LIN {X 0,Y 446.131,Z 914.259,A -85,B 0,C 180,E1 18585.632,E2 18585.632} C_VEL
LIN {X 0,Y 452.831,Z 893.973,A -85,B 0,C 180,E1 18583.695,E2 18583.695} C_VEL
LIN {X 0,Y 459.309,Z 872.522,A -85,B 0,C 180,E1 18581.967,E2 18581.967} C_VEL
LIN {X 0,Y 464.542,Z 853.932,A -85,B 0,C 180,E1 18580.675,E2 18580.675} C_VEL
LIN {X 0,Y 469.911,Z 833.178,A -85,B 0,C 180,E1 18579.43,E2 18579.43} C_VEL
LIN {X 0,Y 475.402,Z 809.084,A -85,B 0,C 180,E1 18578.228,E2 18578.228} C_VEL
LIN {X 0,Y 479.6,Z 787.75,A -85,B 0,C 180,E1 18577.351,E2 18577.351} C_VEL
LIN {X 0,Y 483.367,Z 765.529,A -85,B 0,C 180,E1 18576.603,E2 18576.603} C_VEL
LIN {X 0,Y 487.105,Z 737.581,A -85,B 0,C 180,E1 18575.887,E2 18575.887} C_VEL
LIN {X 0,Y 489.19,Z 714.963,A -85,B 0,C 180,E1 18575.454,E2 18575.454} C_VEL
LIN {X 0,Y 502.118,Z 484.551,A -85,B 0,C 180,E1 18571.853,E2 18571.853} C_VEL
LIN {X 0,Y 505.42,Z 425.189,A -85,B 0,C 180,E1 18570.906,E2 18570.906} C_VEL
LIN {X 0,Y 497.545,Z 411.726,A -85,B 0,C 180,E1 18569.067,E2 18569.067} C_VEL
LIN {X 0,Y 488.892,Z 397.653,A -85,B 0,C 180,E1 18566.872,E2 18566.872} C_VEL
LIN {X 0,Y 478.631,Z 382.114,A -85,B 0,C 180,E1 18563.974,E2 18563.974} C_VEL
LIN {X 0,Y 470.083,Z 371.062,A -85,B 0,C 180,E1 18561.264,E2 18561.264} C_VEL
LIN {X 0,Y 465.83,Z 365.703,A -85,B 0,C 180,E1 18559.759,E2 18559.759} C_VEL
LIN {X 0,Y 461.713,Z 360.509,A -85,B 0,C 180,E1 18558.171,E2 18558.171} C_VEL
LIN {X 0,Y 457.361,Z 355.125,A -85,B 0,C 180,E1 18556.316,E2 18556.316} C_VEL
LIN {X 0,Y 453.894,Z 351.057,A -85,B 0,C 180,E1 18554.675,E2 18554.675} C_VEL
LIN {X 0,Y 452.721,Z 349.402,A -85,B 0,C 180,E1 18554.061,E2 18554.061} C_VEL
LIN {X 0,Y 449.237,Z 345.797,A -85,B 0,C 180,E1 18552.142,E2 18552.142} C_VEL
LIN {X 0,Y 447.81,Z 343.423,A -85,B 0,C 180,E1 18551.201,E2 18551.201} C_VEL
LIN {X 0,Y 444.369,Z 340.419,A -85,B 0,C 180,E1 18548.801,E2 18548.801} C_VEL
LIN {X 0,Y 442.614,Z 337.176,A -85,B 0,C 180,E1 18547.137,E2 18547.137} C_VEL
LIN {X 0,Y 438.09,Z 332.937,A -85,B 0,C 180,E1 18539.346,E2 18539.346} C_VEL
LIN {X 0,Y 438.15,Z 333.065,A -85,B 0,C 180,E1 18536.991,E2 18536.991} C_VEL
LIN {X 0,Y 442.91,Z 337.557,A -85,B 0,C 180,E1 18529.398,E2 18529.398} C_VEL
LIN {X 0,Y 444.805,Z 340.967,A -85,B 0,C 180,E1 18527.669,E2 18527.669} C_VEL
LIN {X 0,Y 448.152,Z 343.843,A -85,B 0,C 180,E1 18525.397,E2 18525.397} C_VEL
LIN {X 0,Y 450.898,Z 347.851,A -85,B 0,C 180,E1 18523.709,E2 18523.709} C_VEL
LIN {X 0,Y 453.392,Z 350.187,A -85,B 0,C 180,E1 18522.414,E2 18522.414} C_VEL
LIN {X 0,Y 456.634,Z 354.467,A -85,B 0,C 180,E1 18520.825,E2 18520.825} C_VEL
LIN {X 0,Y 458.34,Z 356.318,A -85,B 0,C 180,E1 18520.07,E2 18520.07} C_VEL
LIN {X 0,Y 462.075,Z 360.858,A -85,B 0,C 180,E1 18518.509,E2 18518.509} C_VEL
LIN {X 0,Y 467.83,Z 368.146,A -85,B 0,C 180,E1 18516.342,E2 18516.342} C_VEL
LIN {X 0,Y 472.295,Z 373.974,A -85,B 0,C 180,E1 18514.815,E2 18514.815} C_VEL
LIN {X 0,Y 479.579,Z 383.444,A -85,B 0,C 180,E1 18512.563,E2 18512.563} C_VEL
LIN {X 0,Y 489.38,Z 397.087,A -85,B 0,C 180,E1 18509.86,E2 18509.86} C_VEL
LIN {X 0,Y 497.663,Z 409.437,A -85,B 0,C 180,E1 18507.796,E2 18507.796} C_VEL
LIN {X 0,Y 505.573,Z 422.879,A -85,B 0,C 180,E1 18505.951,E2 18505.951} C_VEL
LIN {X 0,Y 493.861,Z 629.815,A -85,B 0,C 180,E1 18502.723,E2 18502.723} C_VEL
LIN {X 0,Y 489.029,Z 714.247,A -85,B 0,C 180,E1 18501.386,E2 18501.386} C_VEL
LIN {X 0,Y 486.062,Z 742.57,A -85,B 0,C 180,E1 18500.783,E2 18500.783} C_VEL
LIN {X 0,Y 483.078,Z 763.5,A -85,B 0,C 180,E1 18500.191,E2 18500.191} C_VEL
LIN {X 0,Y 479.517,Z 784.275,A -85,B 0,C 180,E1 18499.469,E2 18499.469} C_VEL
LIN {X 0,Y 474.318,Z 810.058,A -85,B 0,C 180,E1 18498.357,E2 18498.357} C_VEL
LIN {X 0,Y 469.237,Z 831.534,A -85,B 0,C 180,E1 18497.223,E2 18497.223} C_VEL
LIN {X 0,Y 464.133,Z 851.066,A -85,B 0,C 180,E1 18496.016,E2 18496.016} C_VEL
LIN {X 0,Y 457.617,Z 873.85,A -85,B 0,C 180,E1 18494.362,E2 18494.362} C_VEL
LIN {X 0,Y 451.329,Z 893.778,A -85,B 0,C 180,E1 18492.648,E2 18492.648} C_VEL
LIN {X 0,Y 445.384,Z 911.684,A -85,B 0,C 180,E1 18490.875,E2 18490.875} C_VEL
LIN {X 0,Y 438.182,Z 932.354,A -85,B 0,C 180,E1 18488.492,E2 18488.492} C_VEL
LIN {X 0,Y 432.293,Z 948.557,A -85,B 0,C 180,E1 18486.308,E2 18486.308} C_VEL
LIN {X 0,Y 426.626,Z 963.981,A -85,B 0,C 180,E1 18483.934,E2 18483.934} C_VEL
LIN {X 0,Y 420.149,Z 981.509,A -85,B 0,C 180,E1 18480.781,E2 18480.781} C_VEL
LIN {X 0,Y 415.589,Z 994.103,A -85,B 0,C 180,E1 18478.136,E2 18478.136} C_VEL
LIN {X 0,Y 411.172,Z 1006.966,A -85,B 0,C 180,E1 18475.032,E2 18475.032} C_VEL
LIN {X 0,Y 407.325,Z 1018.86,A -85,B 0,C 180,E1 18471.605,E2 18471.605} C_VEL
LIN {X 0,Y 404.734,Z 1027.798,A -85,B 0,C 180,E1 18468.584,E2 18468.584} C_VEL
LIN {X 0,Y 402.535,Z 1036.804,A -85,B 0,C 180,E1 18464.971,E2 18464.971} C_VEL
LIN {X 0,Y 401.176,Z 1043.635,A -85,B 0,C 180,E1 18461.501,E2 18461.501} C_VEL
LIN {X 0,Y 400.461,Z 1048.425,A -85,B 0,C 180,E1 18458.471,E2 18458.471} C_VEL
LIN {X 0,Y 400.088,Z 1052.26,A -85,B 0,C 180,E1 18455.306,E2 18455.306} C_VEL
LIN {X 0,Y 399.924,Z 1055.14,A -85,B 0,C 180,E1 18451.719,E2 18451.719} C_VEL
LIN {X 0,Y 399.904,Z 1056.343,A -85,B 0,C 180,E1 18448.567,E2 18448.567} C_VEL
LIN {X 0,Y 399.903,Z 1056.481,A -85,B 0,C 180,E1 18447.693,E2 18447.693} C_VEL
LIN {X 0,Y 398.901,Z 1056.59,A -85,B 0,C 180,E1 18446.59,E2 18446.59} C_VEL
LIN {X 0,Y 392.465,Z 1056.003,A -85,B 0,C 180,E1 18443.478,E2 18443.478} C_VEL
LIN {X 0,Y 391.928,Z 1055.619,A -85,B 0,C 180,E1 18442.666,E2 18442.666} C_VEL
LIN {X 0,Y 392.038,Z 1053.632,A -85,B 0,C 180,E1 18439.567,E2 18439.567} C_VEL
LIN {X 0,Y 392.422,Z 1049.847,A -85,B 0,C 180,E1 18435.841,E2 18435.841} C_VEL
LIN {X 0,Y 393.228,Z 1044.792,A -85,B 0,C 180,E1 18432.387,E2 18432.387} C_VEL
LIN {X 0,Y 394.417,Z 1039.146,A -85,B 0,C 180,E1 18429.303,E2 18429.303} C_VEL
LIN {X 0,Y 396.415,Z 1031.684,A -85,B 0,C 180,E1 18425.936,E2 18425.936} C_VEL
LIN {X 0,Y 399.69,Z 1021.249,A -85,B 0,C 180,E1 18422.108,E2 18422.108} C_VEL
LIN {X 0,Y 403.089,Z 1011.528,A -85,B 0,C 180,E1 18419.104,E2 18419.104} C_VEL
LIN {X 0,Y 407.809,Z 999.269,A -85,B 0,C 180,E1 18415.842,E2 18415.842} C_VEL
LIN {X 0,Y 413.485,Z 984.893,A -85,B 0,C 180,E1 18412.63,E2 18412.63} C_VEL
LIN {X 0,Y 418.923,Z 971.568,A -85,B 0,C 180,E1 18410.055,E2 18410.055} C_VEL
LIN {X 0,Y 425.983,Z 954.445,A -85,B 0,C 180,E1 18407.196,E2 18407.196} C_VEL
LIN {X 0,Y 432.891,Z 937.105,A -85,B 0,C 180,E1 18404.744,E2 18404.744} C_VEL
LIN {X 0,Y 439.213,Z 920.922,A -85,B 0,C 180,E1 18402.752,E2 18402.752} C_VEL
LIN {X 0,Y 446.85,Z 900.493,A -85,B 0,C 180,E1 18400.582,E2 18400.582} C_VEL
LIN {X 0,Y 453.657,Z 880.878,A -85,B 0,C 180,E1 18398.819,E2 18398.819} C_VEL
LIN {X 0,Y 459.787,Z 862.035,A -85,B 0,C 180,E1 18397.354,E2 18397.354} C_VEL
LIN {X 0,Y 466.454,Z 839.808,A -85,B 0,C 180,E1 18395.877,E2 18395.877} C_VEL
LIN {X 0,Y 472.255,Z 817.735,A -85,B 0,C 180,E1 18394.659,E2 18394.659} C_VEL
LIN {X 0,Y 476.724,Z 798.729,A -85,B 0,C 180,E1 18393.767,E2 18393.767} C_VEL
LIN {X 0,Y 481.183,Z 777.074,A -85,B 0,C 180,E1 18392.913,E2 18392.913} C_VEL
LIN {X 0,Y 485.71,Z 750.138,A -85,B 0,C 180,E1 18392.076,E2 18392.076} C_VEL
LIN {X 0,Y 488.616,Z 727.847,A -85,B 0,C 180,E1 18391.55,E2 18391.55} C_VEL
LIN {X 0,Y 490.902,Z 702.791,A -85,B 0,C 180,E1 18391.093,E2 18391.093} C_VEL
LIN {X 0,Y 505.255,Z 471.196,A -85,B 0,C 180,E1 18387.473,E2 18387.473} C_VEL
LIN {X 0,Y 507.793,Z 430.464,A -85,B 0,C 180,E1 18386.82,E2 18386.82} C_VEL
LIN {X 0,Y 500.137,Z 417.918,A -85,B 0,C 180,E1 18384.762,E2 18384.762} C_VEL
LIN {X 0,Y 492.623,Z 406.949,A -85,B 0,C 180,E1 18382.558,E2 18382.558} C_VEL
LIN {X 0,Y 485.385,Z 396.927,A -85,B 0,C 180,E1 18380.185,E2 18380.185} C_VEL
LIN {X 0,Y 480.887,Z 391.016,A -85,B 0,C 180,E1 18378.55,E2 18378.55} C_VEL
LIN {X 0,Y 477.714,Z 386.768,A -85,B 0,C 180,E1 18377.291,E2 18377.291} C_VEL
LIN {X 0,Y 474.093,Z 382.002,A -85,B 0,C 180,E1 18375.725,E2 18375.725} C_VEL
LIN {X 0,Y 469.843,Z 376.609,A -85,B 0,C 180,E1 18373.664,E2 18373.664} C_VEL
LIN {X 0,Y 466.423,Z 372.307,A -85,B 0,C 180,E1 18371.751,E2 18371.751} C_VEL
LIN {X 0,Y 465.453,Z 371.035,A -85,B 0,C 180,E1 18371.148,E2 18371.148} C_VEL
LIN {X 0,Y 462.123,Z 367.252,A -85,B 0,C 180,E1 18368.837,E2 18368.837} C_VEL
LIN {X 0,Y 461.146,Z 365.386,A -85,B 0,C 180,E1 18367.977,E2 18367.977} C_VEL
LIN {X 0,Y 457.851,Z 362.35,A -85,B 0,C 180,E1 18364.635,E2 18364.635} C_VEL
LIN {X 0,Y 456.621,Z 359.617,A -85,B 0,C 180,E1 18362.385,E2 18362.385} C_VEL
LIN {X 0,Y 455.677,Z 358.962,A -85,B 0,C 180,E1 18358.365,E2 18358.365} C_VEL
LIN {X 0,Y 456.743,Z 359.705,A -85,B 0,C 180,E1 18354.472,E2 18354.472} C_VEL
LIN {X 0,Y 459.197,Z 364.086,A -85,B 0,C 180,E1 18350.854,E2 18350.854} C_VEL
LIN {X 0,Y 461.418,Z 365.771,A -85,B 0,C 180,E1 18348.88,E2 18348.88} C_VEL
LIN {X 0,Y 464.109,Z 369.819,A -85,B 0,C 180,E1 18346.799,E2 18346.799} C_VEL
LIN {X 0,Y 466.134,Z 371.817,A -85,B 0,C 180,E1 18345.528,E2 18345.528} C_VEL
LIN {X 0,Y 469.371,Z 376.177,A -85,B 0,C 180,E1 18343.668,E2 18343.668} C_VEL
LIN {X 0,Y 470.895,Z 377.833,A -85,B 0,C 180,E1 18342.897,E2 18342.897} C_VEL
LIN {X 0,Y 475.393,Z 383.739,A -85,B 0,C 180,E1 18340.788,E2 18340.788} C_VEL
LIN {X 0,Y 480.025,Z 389.872,A -85,B 0,C 180,E1 18338.878,E2 18338.878} C_VEL
LIN {X 0,Y 484.61,Z 396.005,A -85,B 0,C 180,E1 18337.176,E2 18337.176} C_VEL
LIN {X 0,Y 491.704,Z 406.708,A -85,B 0,C 180,E1 18334.784,E2 18334.784} C_VEL
LIN {X 0,Y 499.013,Z 418.174,A -85,B 0,C 180,E1 18332.59,E2 18332.59} C_VEL
LIN {X 0,Y 507.826,Z 432.949,A -85,B 0,C 180,E1 18330.199,E2 18330.199} C_VEL
LIN {X 0,Y 493.862,Z 655.807,A -85,B 0,C 180,E1 18326.718,E2 18326.718} C_VEL
LIN {X 0,Y 489.698,Z 720.789,A -85,B 0,C 180,E1 18325.679,E2 18325.679} C_VEL
LIN {X 0,Y 486.513,Z 748.326,A -85,B 0,C 180,E1 18325.1,E2 18325.1} C_VEL
LIN {X 0,Y 483.152,Z 769.669,A -85,B 0,C 180,E1 18324.517,E2 18324.517} C_VEL
LIN {X 0,Y 478.792,Z 792.887,A -85,B 0,C 180,E1 18323.717,E2 18323.717} C_VEL
LIN {X 0,Y 473.1,Z 818.082,A -85,B 0,C 180,E1 18322.624,E2 18322.624} C_VEL
LIN {X 0,Y 467.737,Z 838.822,A -85,B 0,C 180,E1 18321.532,E2 18321.532} C_VEL
LIN {X 0,Y 461.508,Z 860.63,A -85,B 0,C 180,E1 18320.179,E2 18320.179} C_VEL
LIN {X 0,Y 454.148,Z 883.618,A -85,B 0,C 180,E1 18318.466,E2 18318.466} C_VEL
LIN {X 0,Y 447.905,Z 901.761,A -85,B 0,C 180,E1 18316.885,E2 18316.885} C_VEL
LIN {X 0,Y 440.681,Z 921.68,A -85,B 0,C 180,E1 18314.882,E2 18314.882} C_VEL
LIN {X 0,Y 433.14,Z 941.135,A -85,B 0,C 180,E1 18312.561,E2 18312.561} C_VEL
LIN {X 0,Y 427.011,Z 956.58,A -85,B 0,C 180,E1 18310.438,E2 18310.438} C_VEL
LIN {X 0,Y 420.13,Z 973.846,A -85,B 0,C 180,E1 18307.709,E2 18307.709} C_VEL
LIN {X 0,Y 413.758,Z 989.517,A -85,B 0,C 180,E1 18304.772,E2 18304.772} C_VEL
LIN {X 0,Y 408.784,Z 1002.114,A -85,B 0,C 180,E1 18302.058,E2 18302.058} C_VEL
LIN {X 0,Y 403.583,Z 1016.015,A -85,B 0,C 180,E1 18298.565,E2 18298.565} C_VEL
LIN {X 0,Y 399.775,Z 1026.875,A -85,B 0,C 180,E1 18295.321,E2 18295.321} C_VEL
LIN {X 0,Y 396.982,Z 1035.848,A -85,B 0,C 180,E1 18292.198,E2 18292.198} C_VEL
LIN {X 0,Y 394.459,Z 1045.402,A -85,B 0,C 180,E1 18288.167,E2 18288.167} C_VEL
LIN {X 0,Y 393.21,Z 1051.386,A -85,B 0,C 180,E1 18285.033,E2 18285.033} C_VEL
LIN {X 0,Y 392.45,Z 1056.21,A -85,B 0,C 180,E1 18281.91,E2 18281.91} C_VEL
LIN {X 0,Y 392.045,Z 1060.472,A -85,B 0,C 180,E1 18278.279,E2 18278.279} C_VEL
LIN {X 0,Y 391.909,Z 1063.031,A -85,B 0,C 180,E1 18274.683,E2 18274.683} C_VEL
LIN {X 0,Y 391.902,Z 1064.068,A -85,B 0,C 180,E1 18271.755,E2 18271.755} C_VEL
LIN {X 0,Y 391.912,Z 1064.138,A -85,B 0,C 180,E1 18268.977,E2 18268.977} C_VEL
LIN {X 0,Y 391.912,Z 1063.308,A -85,B 0,C 180,E1 18266.197,E2 18266.197} C_VEL
LIN {X 0,Y 391.968,Z 1061.457,A -85,B 0,C 180,E1 18263.261,E2 18263.261} C_VEL
LIN {X 0,Y 392.158,Z 1058.434,A -85,B 0,C 180,E1 18260.164,E2 18260.164} C_VEL
LIN {X 0,Y 392.806,Z 1053.089,A -85,B 0,C 180,E1 18256.306,E2 18256.306} C_VEL
LIN {X 0,Y 393.863,Z 1047.064,A -85,B 0,C 180,E1 18253.026,E2 18253.026} C_VEL
LIN {X 0,Y 395.366,Z 1040.429,A -85,B 0,C 180,E1 18250.037,E2 18250.037} C_VEL
LIN {X 0,Y 397.97,Z 1030.979,A -85,B 0,C 180,E1 18246.454,E2 18246.454} C_VEL
LIN {X 0,Y 401.376,Z 1019.976,A -85,B 0,C 180,E1 18243.039,E2 18243.039} C_VEL
LIN {X 0,Y 404.921,Z 1009.552,A -85,B 0,C 180,E1 18240.242,E2 18240.242} C_VEL
LIN {X 0,Y 409.991,Z 995.753,A -85,B 0,C 180,E1 18237.03,E2 18237.03} C_VEL
LIN {X 0,Y 415.607,Z 980.582,A -85,B 0,C 180,E1 18234.054,E2 18234.054} C_VEL
LIN {X 0,Y 420.867,Z 966.706,A -85,B 0,C 180,E1 18231.678,E2 18231.678} C_VEL
LIN {X 0,Y 427.585,Z 949.121,A -85,B 0,C 180,E1 18229.054,E2 18229.054} C_VEL
LIN {X 0,Y 434.403,Z 930.424,A -85,B 0,C 180,E1 18226.692,E2 18226.692} C_VEL
LIN {X 0,Y 440.243,Z 913.957,A -85,B 0,C 180,E1 18224.878,E2 18224.878} C_VEL
LIN {X 0,Y 447.095,Z 893.834,A -85,B 0,C 180,E1 18222.946,E2 18222.946} C_VEL
LIN {X 0,Y 453.756,Z 872.421,A -85,B 0,C 180,E1 18221.214,E2 18221.214} C_VEL
LIN {X 0,Y 459.049,Z 854.175,A -85,B 0,C 180,E1 18219.94,E2 18219.94} C_VEL
LIN {X 0,Y 464.488,Z 833.744,A -85,B 0,C 180,E1 18218.708,E2 18218.708} C_VEL
LIN {X 0,Y 470.469,Z 808.208,A -85,B 0,C 180,E1 18217.433,E2 18217.433} C_VEL
LIN {X 0,Y 474.742,Z 786.949,A -85,B 0,C 180,E1 18216.564,E2 18216.564} C_VEL
LIN {X 0,Y 478.746,Z 763.73,A -85,B 0,C 180,E1 18215.789,E2 18215.789} C_VEL
LIN {X 0,Y 482.363,Z 736.862,A -85,B 0,C 180,E1 18215.114,E2 18215.114} C_VEL
LIN {X 0,Y 484.457,Z 714.471,A -85,B 0,C 180,E1 18214.686,E2 18214.686} C_VEL
LIN {X 0,Y 497.803,Z 483.887,A -85,B 0,C 180,E1 18211.07,E2 18211.07} C_VEL
LIN {X 0,Y 500.96,Z 429.227,A -85,B 0,C 180,E1 18210.197,E2 18210.197} C_VEL
LIN {X 0,Y 491.432,Z 413.006,A -85,B 0,C 180,E1 18207.87,E2 18207.87} C_VEL
LIN {X 0,Y 483.386,Z 400.09,A -85,B 0,C 180,E1 18205.714,E2 18205.714} C_VEL
LIN {X 0,Y 475.776,Z 388.58,A -85,B 0,C 180,E1 18203.469,E2 18203.469} C_VEL
LIN {X 0,Y 468.088,Z 378.415,A -85,B 0,C 180,E1 18200.965,E2 18200.965} C_VEL
LIN {X 0,Y 463.74,Z 372.888,A -85,B 0,C 180,E1 18199.393,E2 18199.393} C_VEL
LIN {X 0,Y 459.847,Z 367.901,A -85,B 0,C 180,E1 18197.854,E2 18197.854} C_VEL
LIN {X 0,Y 455.606,Z 362.601,A -85,B 0,C 180,E1 18196.004,E2 18196.004} C_VEL
LIN {X 0,Y 452.077,Z 358.219,A -85,B 0,C 180,E1 18194.277,E2 18194.277} C_VEL
LIN {X 0,Y 451.026,Z 356.927,A -85,B 0,C 180,E1 18193.722,E2 18193.722} C_VEL
LIN {X 0,Y 447.649,Z 353.179,A -85,B 0,C 180,E1 18191.793,E2 18191.793} C_VEL
LIN {X 0,Y 446.436,Z 351.192,A -85,B 0,C 180,E1 18190.975,E2 18190.975} C_VEL
LIN {X 0,Y 443.006,Z 347.999,A -85,B 0,C 180,E1 18188.502,E2 18188.502} C_VEL
LIN {X 0,Y 441.501,Z 345.069,A -85,B 0,C 180,E1 18187.025,E2 18187.025} C_VEL
LIN {X 0,Y 437.114,Z 340.88,A -85,B 0,C 180,E1 18179.345,E2 18179.345} C_VEL
LIN {X 0,Y 437.175,Z 341.01,A -85,B 0,C 180,E1 18176.985,E2 18176.985} C_VEL
LIN {X 0,Y 441.727,Z 345.427,A -85,B 0,C 180,E1 18169.567,E2 18169.567} C_VEL
LIN {X 0,Y 443.835,Z 349.051,A -85,B 0,C 180,E1 18167.642,E2 18167.642} C_VEL
LIN {X 0,Y 446.875,Z 351.769,A -85,B 0,C 180,E1 18165.553,E2 18165.553} C_VEL
LIN {X 0,Y 449.712,Z 355.773,A -85,B 0,C 180,E1 18163.797,E2 18163.797} C_VEL
LIN {X 0,Y 451.823,Z 357.76,A -85,B 0,C 180,E1 18162.683,E2 18162.683} C_VEL
LIN {X 0,Y 455.276,Z 362.29,A -85,B 0,C 180,E1 18160.965,E2 18160.965} C_VEL
LIN {X 0,Y 456.822,Z 364.121,A -85,B 0,C 180,E1 18160.264,E2 18160.264} C_VEL
LIN {X 0,Y 461.528,Z 369.973,A -85,B 0,C 180,E1 18158.289,E2 18158.289} C_VEL
LIN {X 0,Y 465.963,Z 375.643,A -85,B 0,C 180,E1 18156.61,E2 18156.61} C_VEL
LIN {X 0,Y 470.369,Z 381.482,A -85,B 0,C 180,E1 18155.075,E2 18155.075} C_VEL
LIN {X 0,Y 477.565,Z 391.013,A -85,B 0,C 180,E1 18152.809,E2 18152.809} C_VEL
LIN {X 0,Y 486.753,Z 403.987,A -85,B 0,C 180,E1 18150.224,E2 18150.224} C_VEL
LIN {X 0,Y 494.926,Z 416.359,A -85,B 0,C 180,E1 18148.143,E2 18148.143} C_VEL
LIN {X 0,Y 501.078,Z 427.113,A -85,B 0,C 180,E1 18146.66,E2 18146.66} C_VEL
LIN {X 0,Y 488.955,Z 634.954,A -85,B 0,C 180,E1 18143.407,E2 18143.407} C_VEL
LIN {X 0,Y 484.241,Z 714.579,A -85,B 0,C 180,E1 18142.14,E2 18142.14} C_VEL
LIN {X 0,Y 481.19,Z 742.87,A -85,B 0,C 180,E1 18141.535,E2 18141.535} C_VEL
LIN {X 0,Y 478.158,Z 763.597,A -85,B 0,C 180,E1 18140.949,E2 18140.949} C_VEL
LIN {X 0,Y 474.38,Z 785.067,A -85,B 0,C 180,E1 18140.2,E2 18140.2} C_VEL
LIN {X 0,Y 468.781,Z 811.803,A -85,B 0,C 180,E1 18139.031,E2 18139.031} C_VEL
LIN {X 0,Y 463.82,Z 832.15,A -85,B 0,C 180,E1 18137.947,E2 18137.947} C_VEL
LIN {X 0,Y 458.345,Z 852.473,A -85,B 0,C 180,E1 18136.68,E2 18136.68} C_VEL
LIN {X 0,Y 451.182,Z 876.452,A -85,B 0,C 180,E1 18134.899,E2 18134.899} C_VEL
LIN {X 0,Y 445.054,Z 895.256,A -85,B 0,C 180,E1 18133.254,E2 18133.254} C_VEL
LIN {X 0,Y 438.462,Z 914.469,A -85,B 0,C 180,E1 18131.314,E2 18131.314} C_VEL
LIN {X 0,Y 431.168,Z 934.445,A -85,B 0,C 180,E1 18128.936,E2 18128.936} C_VEL
LIN {X 0,Y 425.394,Z 949.785,A -85,B 0,C 180,E1 18126.825,E2 18126.825} C_VEL
LIN {X 0,Y 418.888,Z 966.933,A -85,B 0,C 180,E1 18124.121,E2 18124.121} C_VEL
LIN {X 0,Y 412.853,Z 982.489,A -85,B 0,C 180,E1 18121.217,E2 18121.217} C_VEL
LIN {X 0,Y 408.151,Z 994.975,A -85,B 0,C 180,E1 18118.536,E2 18118.536} C_VEL
LIN {X 0,Y 403.336,Z 1008.405,A -85,B 0,C 180,E1 18115.196,E2 18115.196} C_VEL
LIN {X 0,Y 399.587,Z 1019.513,A -85,B 0,C 180,E1 18111.891,E2 18111.891} C_VEL
LIN {X 0,Y 396.901,Z 1028.385,A -85,B 0,C 180,E1 18108.812,E2 18108.812} C_VEL
LIN {X 0,Y 394.541,Z 1037.562,A -85,B 0,C 180,E1 18104.981,E2 18104.981} C_VEL
LIN {X 0,Y 393.208,Z 1044.033,A -85,B 0,C 180,E1 18101.589,E2 18101.589} C_VEL
LIN {X 0,Y 392.47,Z 1048.763,A -85,B 0,C 180,E1 18098.497,E2 18098.497} C_VEL
LIN {X 0,Y 392.06,Z 1053.002,A -85,B 0,C 180,E1 18094.828,E2 18094.828} C_VEL
LIN {X 0,Y 391.923,Z 1055.438,A -85,B 0,C 180,E1 18091.316,E2 18091.316} C_VEL
LIN {X 0,Y 391.904,Z 1056.449,A -85,B 0,C 180,E1 18088.392,E2 18088.392} C_VEL
LIN {X 0,Y 391.908,Z 1056.512,A -85,B 0,C 180,E1 18085.61,E2 18085.61} C_VEL
LIN {X 0,Y 391.934,Z 1055.688,A -85,B 0,C 180,E1 18082.819,E2 18082.819} C_VEL
LIN {X 0,Y 391.928,Z 1055.619,A -85,B 0,C 180,E1 18082.666,E2 18082.666} C_VEL
LIN {X 0,Y 390.935,Z 1055.128,A -85,B 0,C 180,E1 18081.542,E2 18081.542} C_VEL
LIN {X 0,Y 384.638,Z 1052.892,A -85,B 0,C 180,E1 18078.378,E2 18078.378} C_VEL
LIN {X 0,Y 384.191,Z 1052.05,A -85,B 0,C 180,E1 18077.557,E2 18077.557} C_VEL
LIN {X 0,Y 384.687,Z 1048.427,A -85,B 0,C 180,E1 18074.471,E2 18074.471} C_VEL
LIN {X 0,Y 385.611,Z 1043.532,A -85,B 0,C 180,E1 18071.244,E2 18071.244} C_VEL
LIN {X 0,Y 387.471,Z 1036.151,A -85,B 0,C 180,E1 18067.387,E2 18067.387} C_VEL
LIN {X 0,Y 390.059,Z 1027.614,A -85,B 0,C 180,E1 18063.838,E2 18063.838} C_VEL
LIN {X 0,Y 393.101,Z 1018.845,A -85,B 0,C 180,E1 18060.746,E2 18060.746} C_VEL
LIN {X 0,Y 397.824,Z 1006.581,A -85,B 0,C 180,E1 18057.085,E2 18057.085} C_VEL
LIN {X 0,Y 402.873,Z 994.132,A -85,B 0,C 180,E1 18053.97,E2 18053.97} C_VEL
LIN {X 0,Y 408.322,Z 981.262,A -85,B 0,C 180,E1 18051.179,E2 18051.179} C_VEL
LIN {X 0,Y 415.587,Z 964.18,A -85,B 0,C 180,E1 18048.021,E2 18048.021} C_VEL
LIN {X 0,Y 421.937,Z 949.133,A -85,B 0,C 180,E1 18045.647,E2 18045.647} C_VEL
LIN {X 0,Y 428.929,Z 932.323,A -85,B 0,C 180,E1 18043.339,E2 18043.339} C_VEL
LIN {X 0,Y 436.989,Z 911.98,A -85,B 0,C 180,E1 18040.968,E2 18040.968} C_VEL
LIN {X 0,Y 443.464,Z 894.72,A -85,B 0,C 180,E1 18039.241,E2 18039.241} C_VEL
LIN {X 0,Y 450.313,Z 875.392,A -85,B 0,C 180,E1 18037.562,E2 18037.562} C_VEL
LIN {X 0,Y 457.777,Z 852.281,A -85,B 0,C 180,E1 18035.87,E2 18035.87} C_VEL
LIN {X 0,Y 463.611,Z 832.274,A -85,B 0,C 180,E1 18034.635,E2 18034.635} C_VEL
LIN {X 0,Y 469.347,Z 810.445,A -85,B 0,C 180,E1 18033.489,E2 18033.489} C_VEL
LIN {X 0,Y 475.126,Z 784.661,A -85,B 0,C 180,E1 18032.391,E2 18032.391} C_VEL
LIN {X 0,Y 479.205,Z 763.06,A -85,B 0,C 180,E1 18031.652,E2 18031.652} C_VEL
LIN {X 0,Y 482.663,Z 741.008,A -85,B 0,C 180,E1 18031.049,E2 18031.049} C_VEL
LIN {X 0,Y 485.737,Z 713.616,A -85,B 0,C 180,E1 18030.484,E2 18030.484} C_VEL
LIN {X 0,Y 494.66,Z 574.998,A -85,B 0,C 180,E1 18028.295,E2 18028.295} C_VEL
LIN {X 0,Y 503.713,Z 434.872,A -85,B 0,C 180,E1 18026.084,E2 18026.084} C_VEL
LIN {X 0,Y 496.679,Z 423.301,A -85,B 0,C 180,E1 18024.121,E2 18024.121} C_VEL
LIN {X 0,Y 487.17,Z 409.41,A -85,B 0,C 180,E1 18021.176,E2 18021.176} C_VEL
LIN {X 0,Y 480.051,Z 399.679,A -85,B 0,C 180,E1 18018.646,E2 18018.646} C_VEL
LIN {X 0,Y 475.749,Z 393.971,A -85,B 0,C 180,E1 18016.923,E2 18016.923} C_VEL
LIN {X 0,Y 472.334,Z 389.412,A -85,B 0,C 180,E1 18015.407,E2 18015.407} C_VEL
LIN {X 0,Y 468.287,Z 384.193,A -85,B 0,C 180,E1 18013.395,E2 18013.395} C_VEL
LIN {X 0,Y 464.947,Z 379.841,A -85,B 0,C 180,E1 18011.474,E2 18011.474} C_VEL
LIN {X 0,Y 463.891,Z 378.599,A -85,B 0,C 180,E1 18010.808,E2 18010.808} C_VEL
LIN {X 0,Y 460.764,Z 374.802,A -85,B 0,C 180,E1 18008.549,E2 18008.549} C_VEL
LIN {X 0,Y 459.873,Z 373.176,A -85,B 0,C 180,E1 18007.747,E2 18007.747} C_VEL
LIN {X 0,Y 456.694,Z 370.084,A -85,B 0,C 180,E1 18004.395,E2 18004.395} C_VEL
LIN {X 0,Y 455.586,Z 367.512,A -85,B 0,C 180,E1 18002.264,E2 18002.264} C_VEL
LIN {X 0,Y 454.712,Z 366.903,A -85,B 0,C 180,E1 17998.11,E2 17998.11} C_VEL
LIN {X 0,Y 455.706,Z 367.603,A -85,B 0,C 180,E1 17994.586,E2 17994.586} C_VEL
LIN {X 0,Y 458.107,Z 371.967,A -85,B 0,C 180,E1 17990.958,E2 17990.958} C_VEL
LIN {X 0,Y 460.221,Z 373.622,A -85,B 0,C 180,E1 17989.041,E2 17989.041} C_VEL
LIN {X 0,Y 462.96,Z 377.717,A -85,B 0,C 180,E1 17986.893,E2 17986.893} C_VEL
LIN {X 0,Y 464.765,Z 379.542,A -85,B 0,C 180,E1 17985.739,E2 17985.739} C_VEL
LIN {X 0,Y 468.065,Z 383.985,A -85,B 0,C 180,E1 17983.813,E2 17983.813} C_VEL
LIN {X 0,Y 469.559,Z 385.756,A -85,B 0,C 180,E1 17983.038,E2 17983.038} C_VEL
LIN {X 0,Y 473.765,Z 391.33,A -85,B 0,C 180,E1 17981.033,E2 17981.033} C_VEL
LIN {X 0,Y 478.315,Z 397.448,A -85,B 0,C 180,E1 17979.119,E2 17979.119} C_VEL
LIN {X 0,Y 482.918,Z 403.701,A -85,B 0,C 180,E1 17977.381,E2 17977.381} C_VEL
LIN {X 0,Y 491.664,Z 417.188,A -85,B 0,C 180,E1 17974.428,E2 17974.428} C_VEL
LIN {X 0,Y 498.732,Z 428.868,A -85,B 0,C 180,E1 17972.314,E2 17972.314} C_VEL
LIN {X 0,Y 503.735,Z 437.492,A -85,B 0,C 180,E1 17970.931,E2 17970.931} C_VEL
LIN {X 0,Y 489.337,Z 660.875,A -85,B 0,C 180,E1 17967.435,E2 17967.435} C_VEL
LIN {X 0,Y 485.33,Z 721.242,A -85,B 0,C 180,E1 17966.465,E2 17966.465} C_VEL
LIN {X 0,Y 482.074,Z 748.505,A -85,B 0,C 180,E1 17965.89,E2 17965.89} C_VEL
LIN {X 0,Y 478.634,Z 769.802,A -85,B 0,C 180,E1 17965.309,E2 17965.309} C_VEL
LIN {X 0,Y 474.242,Z 792.619,A -85,B 0,C 180,E1 17964.524,E2 17964.524} C_VEL
LIN {X 0,Y 468.259,Z 818.421,A -85,B 0,C 180,E1 17963.406,E2 17963.406} C_VEL
LIN {X 0,Y 462.868,Z 838.734,A -85,B 0,C 180,E1 17962.335,E2 17962.335} C_VEL
LIN {X 0,Y 456.63,Z 859.991,A -85,B 0,C 180,E1 17961.018,E2 17961.018} C_VEL
LIN {X 0,Y 449.047,Z 883.08,A -85,B 0,C 180,E1 17959.304,E2 17959.304} C_VEL
LIN {X 0,Y 442.601,Z 901.262,A -85,B 0,C 180,E1 17957.719,E2 17957.719} C_VEL
LIN {X 0,Y 435.582,Z 920.009,A -85,B 0,C 180,E1 17955.836,E2 17955.836} C_VEL
LIN {X 0,Y 427.41,Z 940.495,A -85,B 0,C 180,E1 17953.407,E2 17953.407} C_VEL
LIN {X 0,Y 421.129,Z 955.745,A -85,B 0,C 180,E1 17951.304,E2 17951.304} C_VEL
LIN {X 0,Y 414.256,Z 972.255,A -85,B 0,C 180,E1 17948.693,E2 17948.693} C_VEL
LIN {X 0,Y 407.451,Z 988.389,A -85,B 0,C 180,E1 17945.68,E2 17945.68} C_VEL
LIN {X 0,Y 402.278,Z 1000.879,A -85,B 0,C 180,E1 17942.979,E2 17942.979} C_VEL
LIN {X 0,Y 397.036,Z 1014.14,A -85,B 0,C 180,E1 17939.675,E2 17939.675} C_VEL
LIN {X 0,Y 392.606,Z 1025.955,A -85,B 0,C 180,E1 17936.142,E2 17936.142} C_VEL
LIN {X 0,Y 389.714,Z 1034.62,A -85,B 0,C 180,E1 17933.113,E2 17933.113} C_VEL
LIN {X 0,Y 387.147,Z 1043.501,A -85,B 0,C 180,E1 17929.461,E2 17929.461} C_VEL
LIN {X 0,Y 385.411,Z 1050.837,A -85,B 0,C 180,E1 17925.653,E2 17925.653} C_VEL
LIN {X 0,Y 384.559,Z 1055.748,A -85,B 0,C 180,E1 17922.463,E2 17922.463} C_VEL
LIN {X 0,Y 384.108,Z 1059.528,A -85,B 0,C 180,E1 17919.288,E2 17919.288} C_VEL
LIN {X 0,Y 383.926,Z 1062.541,A -85,B 0,C 180,E1 17915.68,E2 17915.68} C_VEL
LIN {X 0,Y 383.908,Z 1063.947,A -85,B 0,C 180,E1 17912.09,E2 17912.09} C_VEL
LIN {X 0,Y 383.912,Z 1064.08,A -85,B 0,C 180,E1 17909.105,E2 17909.105} C_VEL
LIN {X 0,Y 383.912,Z 1063.288,A -85,B 0,C 180,E1 17906.267,E2 17906.267} C_VEL
LIN {X 0,Y 383.967,Z 1061.476,A -85,B 0,C 180,E1 17903.27,E2 17903.27} C_VEL
LIN {X 0,Y 384.15,Z 1058.653,A -85,B 0,C 180,E1 17900.26,E2 17900.26} C_VEL
LIN {X 0,Y 384.73,Z 1053.961,A -85,B 0,C 180,E1 17896.626,E2 17896.626} C_VEL
LIN {X 0,Y 385.884,Z 1047.537,A -85,B 0,C 180,E1 17892.969,E2 17892.969} C_VEL
LIN {X 0,Y 387.514,Z 1040.648,A -85,B 0,C 180,E1 17889.772,E2 17889.772} C_VEL
LIN {X 0,Y 389.968,Z 1032.06,A -85,B 0,C 180,E1 17886.423,E2 17886.423} C_VEL
LIN {X 0,Y 393.78,Z 1020.327,A -85,B 0,C 180,E1 17882.639,E2 17882.639} C_VEL
LIN {X 0,Y 397.476,Z 1009.951,A -85,B 0,C 180,E1 17879.794,E2 17879.794} C_VEL
LIN {X 0,Y 402.181,Z 997.581,A -85,B 0,C 180,E1 17876.842,E2 17876.842} C_VEL
LIN {X 0,Y 408.265,Z 981.922,A -85,B 0,C 180,E1 17873.652,E2 17873.652} C_VEL
LIN {X 0,Y 414.007,Z 967.326,A -85,B 0,C 180,E1 17871.102,E2 17871.102} C_VEL
LIN {X 0,Y 420.653,Z 950.528,A -85,B 0,C 180,E1 17868.548,E2 17868.548} C_VEL
LIN {X 0,Y 427.975,Z 931.264,A -85,B 0,C 180,E1 17866.062,E2 17866.062} C_VEL
LIN {X 0,Y 433.986,Z 914.882,A -85,B 0,C 180,E1 17864.231,E2 17864.231} C_VEL
LIN {X 0,Y 440.396,Z 896.628,A -85,B 0,C 180,E1 17862.448,E2 17862.448} C_VEL
LIN {X 0,Y 447.955,Z 873.401,A -85,B 0,C 180,E1 17860.523,E2 17860.523} C_VEL
LIN {X 0,Y 453.637,Z 854.401,A -85,B 0,C 180,E1 17859.187,E2 17859.187} C_VEL
LIN {X 0,Y 459.14,Z 834.306,A -85,B 0,C 180,E1 17857.97,E2 17857.97} C_VEL
LIN {X 0,Y 465.339,Z 808.655,A -85,B 0,C 180,E1 17856.68,E2 17856.68} C_VEL
LIN {X 0,Y 469.736,Z 787.379,A -85,B 0,C 180,E1 17855.806,E2 17855.806} C_VEL
LIN {X 0,Y 473.717,Z 764.932,A -85,B 0,C 180,E1 17855.052,E2 17855.052} C_VEL
LIN {X 0,Y 477.582,Z 737.291,A -85,B 0,C 180,E1 17854.349,E2 17854.349} C_VEL
LIN {X 0,Y 479.756,Z 714.738,A -85,B 0,C 180,E1 17853.917,E2 17853.917} C_VEL
LIN {X 0,Y 493.498,Z 484.634,A -85,B 0,C 180,E1 17850.295,E2 17850.295} C_VEL
LIN {X 0,Y 496.518,Z 433.224,A -85,B 0,C 180,E1 17849.464,E2 17849.464} C_VEL
LIN {X 0,Y 485.524,Z 414.465,A -85,B 0,C 180,E1 17846.647,E2 17846.647} C_VEL
LIN {X 0,Y 476.122,Z 399.681,A -85,B 0,C 180,E1 17843.944,E2 17843.944} C_VEL
LIN {X 0,Y 472.423,Z 394.305,A -85,B 0,C 180,E1 17842.788,E2 17842.788} C_VEL
LIN {X 0,Y 465.609,Z 385.181,A -85,B 0,C 180,E1 17840.49,E2 17840.49} C_VEL
LIN {X 0,Y 461.67,Z 380.068,A -85,B 0,C 180,E1 17839.024,E2 17839.024} C_VEL
LIN {X 0,Y 457.996,Z 375.289,A -85,B 0,C 180,E1 17837.535,E2 17837.535} C_VEL
LIN {X 0,Y 453.933,Z 370.132,A -85,B 0,C 180,E1 17835.72,E2 17835.72} C_VEL
LIN {X 0,Y 450.392,Z 365.571,A -85,B 0,C 180,E1 17833.938,E2 17833.938} C_VEL
LIN {X 0,Y 446.079,Z 360.557,A -85,B 0,C 180,E1 17831.442,E2 17831.442} C_VEL
LIN {X 0,Y 445.07,Z 358.954,A -85,B 0,C 180,E1 17830.747,E2 17830.747} C_VEL
LIN {X 0,Y 441.655,Z 355.574,A -85,B 0,C 180,E1 17828.2,E2 17828.2} C_VEL
LIN {X 0,Y 440.252,Z 352.901,A -85,B 0,C 180,E1 17826.783,E2 17826.783} C_VEL
LIN {X 0,Y 436.138,Z 348.822,A -85,B 0,C 180,E1 17819.343,E2 17819.343} C_VEL
LIN {X 0,Y 436.2,Z 348.956,A -85,B 0,C 180,E1 17816.978,E2 17816.978} C_VEL
LIN {X 0,Y 440.549,Z 353.287,A -85,B 0,C 180,E1 17809.737,E2 17809.737} C_VEL
LIN {X 0,Y 442.702,Z 356.946,A -85,B 0,C 180,E1 17807.742,E2 17807.742} C_VEL
LIN {X 0,Y 445.515,Z 359.502,A -85,B 0,C 180,E1 17805.773,E2 17805.773} C_VEL
LIN {X 0,Y 448.527,Z 363.69,A -85,B 0,C 180,E1 17803.886,E2 17803.886} C_VEL
LIN {X 0,Y 450.376,Z 365.526,A -85,B 0,C 180,E1 17802.892,E2 17802.892} C_VEL
LIN {X 0,Y 453.921,Z 370.11,A -85,B 0,C 180,E1 17801.106,E2 17801.106} C_VEL
LIN {X 0,Y 459.737,Z 377.454,A -85,B 0,C 180,E1 17798.569,E2 17798.569} C_VEL
LIN {X 0,Y 464.105,Z 383.137,A -85,B 0,C 180,E1 17796.88,E2 17796.88} C_VEL
LIN {X 0,Y 468.709,Z 389.33,A -85,B 0,C 180,E1 17795.25,E2 17795.25} C_VEL
LIN {X 0,Y 476.117,Z 399.345,A -85,B 0,C 180,E1 17792.889,E2 17792.889} C_VEL
LIN {X 0,Y 484.745,Z 411.808,A -85,B 0,C 180,E1 17790.429,E2 17790.429} C_VEL
LIN {X 0,Y 492.314,Z 423.447,A -85,B 0,C 180,E1 17788.467,E2 17788.467} C_VEL
LIN {X 0,Y 496.668,Z 431.259,A -85,B 0,C 180,E1 17787.384,E2 17787.384} C_VEL
LIN {X 0,Y 484.103,Z 640.32,A -85,B 0,C 180,E1 17784.103,E2 17784.103} C_VEL
LIN {X 0,Y 479.546,Z 714.809,A -85,B 0,C 180,E1 17782.911,E2 17782.911} C_VEL
LIN {X 0,Y 476.421,Z 743.041,A -85,B 0,C 180,E1 17782.306,E2 17782.306} C_VEL
LIN {X 0,Y 473.313,Z 763.754,A -85,B 0,C 180,E1 17781.721,E2 17781.721} C_VEL
LIN {X 0,Y 469.4,Z 785.429,A -85,B 0,C 180,E1 17780.963,E2 17780.963} C_VEL
LIN {X 0,Y 463.846,Z 811.309,A -85,B 0,C 180,E1 17779.833,E2 17779.833} C_VEL
LIN {X 0,Y 458.475,Z 832.773,A -85,B 0,C 180,E1 17778.688,E2 17778.688} C_VEL
LIN {X 0,Y 452.621,Z 853.881,A -85,B 0,C 180,E1 17777.36,E2 17777.36} C_VEL
LIN {X 0,Y 445.409,Z 877.171,A -85,B 0,C 180,E1 17775.609,E2 17775.609} C_VEL
LIN {X 0,Y 439.195,Z 895.664,A -85,B 0,C 180,E1 17773.977,E2 17773.977} C_VEL
LIN {X 0,Y 431.974,Z 916.071,A -85,B 0,C 180,E1 17771.893,E2 17771.893} C_VEL
LIN {X 0,Y 424.666,Z 935.28,A -85,B 0,C 180,E1 17769.561,E2 17769.561} C_VEL
LIN {X 0,Y 418.532,Z 951.011,A -85,B 0,C 180,E1 17767.359,E2 17767.359} C_VEL
LIN {X 0,Y 411.5,Z 968.75,A -85,B 0,C 180,E1 17764.482,E2 17764.482} C_VEL
LIN {X 0,Y 405.798,Z 982.932,A -85,B 0,C 180,E1 17761.779,E2 17761.779} C_VEL
LIN {X 0,Y 400.969,Z 995.22,A -85,B 0,C 180,E1 17759.095,E2 17759.095} C_VEL
LIN {X 0,Y 396,Z 1008.48,A -85,B 0,C 180,E1 17755.74,E2 17755.74} C_VEL
LIN {X 0,Y 392.159,Z 1019.262,A -85,B 0,C 180,E1 17752.486,E2 17752.486} C_VEL
LIN {X 0,Y 389.424,Z 1027.773,A -85,B 0,C 180,E1 17749.499,E2 17749.499} C_VEL
LIN {X 0,Y 386.935,Z 1036.824,A -85,B 0,C 180,E1 17745.743,E2 17745.743} C_VEL
LIN {X 0,Y 385.383,Z 1043.678,A -85,B 0,C 180,E1 17742.131,E2 17742.131} C_VEL
LIN {X 0,Y 384.557,Z 1048.489,A -85,B 0,C 180,E1 17738.975,E2 17738.975} C_VEL
LIN {X 0,Y 384.116,Z 1052.344,A -85,B 0,C 180,E1 17735.677,E2 17735.677} C_VEL
LIN {X 0,Y 383.932,Z 1055.265,A -85,B 0,C 180,E1 17731.94,E2 17731.94} C_VEL
LIN {X 0,Y 383.906,Z 1056.488,A -85,B 0,C 180,E1 17728.657,E2 17728.657} C_VEL
LIN {X 0,Y 383.908,Z 1056.606,A -85,B 0,C 180,E1 17725.668,E2 17725.668} C_VEL
LIN {X 0,Y 383.935,Z 1055.816,A -85,B 0,C 180,E1 17722.819,E2 17722.819} C_VEL
LIN {X 0,Y 384.026,Z 1054.019,A -85,B 0,C 180,E1 17719.802,E2 17719.802} C_VEL
LIN {X 0,Y 384.191,Z 1052.05,A -85,B 0,C 180,E1 17717.557,E2 17717.557} C_VEL
LIN {X 0,Y 383.344,Z 1050.906,A -85,B 0,C 180,E1 17716.418,E2 17716.418} C_VEL
LIN {X 0,Y 377.603,Z 1047.379,A -85,B 0,C 180,E1 17713.285,E2 17713.285} C_VEL
LIN {X 0,Y 377.243,Z 1046.031,A -85,B 0,C 180,E1 17712.379,E2 17712.379} C_VEL
LIN {X 0,Y 378.716,Z 1039.791,A -85,B 0,C 180,E1 17708.749,E2 17708.749} C_VEL
LIN {X 0,Y 380.737,Z 1032.952,A -85,B 0,C 180,E1 17705.485,E2 17705.485} C_VEL
LIN {X 0,Y 384.221,Z 1023.01,A -85,B 0,C 180,E1 17701.56,E2 17701.56} C_VEL
LIN {X 0,Y 388.277,Z 1012.451,A -85,B 0,C 180,E1 17698.135,E2 17698.135} C_VEL
LIN {X 0,Y 392.895,Z 1001.435,A -85,B 0,C 180,E1 17695.068,E2 17695.068} C_VEL
LIN {X 0,Y 399.569,Z 986.099,A -85,B 0,C 180,E1 17691.457,E2 17691.457} C_VEL
LIN {X 0,Y 405.562,Z 972.588,A -85,B 0,C 180,E1 17688.761,E2 17688.761} C_VEL
LIN {X 0,Y 412.598,Z 956.824,A -85,B 0,C 180,E1 17686.034,E2 17686.034} C_VEL
LIN {X 0,Y 420.199,Z 939.204,A -85,B 0,C 180,E1 17683.448,E2 17683.448} C_VEL
LIN {X 0,Y 427.065,Z 922.814,A -85,B 0,C 180,E1 17681.376,E2 17681.376} C_VEL
LIN {X 0,Y 434.489,Z 904.383,A -85,B 0,C 180,E1 17679.355,E2 17679.355} C_VEL
LIN {X 0,Y 442.644,Z 882.529,A -85,B 0,C 180,E1 17677.332,E2 17677.332} C_VEL
LIN {X 0,Y 449.094,Z 863.893,A -85,B 0,C 180,E1 17675.862,E2 17675.862} C_VEL
LIN {X 0,Y 455.587,Z 843.623,A -85,B 0,C 180,E1 17674.489,E2 17674.489} C_VEL
LIN {X 0,Y 462.521,Z 819.067,A -85,B 0,C 180,E1 17673.102,E2 17673.102} C_VEL
LIN {X 0,Y 467.329,Z 799.757,A -85,B 0,C 180,E1 17672.192,E2 17672.192} C_VEL
LIN {X 0,Y 471.716,Z 779.608,A -85,B 0,C 180,E1 17671.389,E2 17671.389} C_VEL
LIN {X 0,Y 476.446,Z 753.778,A -85,B 0,C 180,E1 17670.561,E2 17670.561} C_VEL
LIN {X 0,Y 479.838,Z 729.417,A -85,B 0,C 180,E1 17669.978,E2 17669.978} C_VEL
LIN {X 0,Y 482.097,Z 706.648,A -85,B 0,C 180,E1 17669.555,E2 17669.555} C_VEL
LIN {X 0,Y 497.394,Z 474.9,A -85,B 0,C 180,E1 17665.916,E2 17665.916} C_VEL
LIN {X 0,Y 499.766,Z 439.404,A -85,B 0,C 180,E1 17665.351,E2 17665.351} C_VEL
LIN {X 0,Y 493.365,Z 428.928,A -85,B 0,C 180,E1 17663.5,E2 17663.5} C_VEL
LIN {X 0,Y 484.676,Z 416.117,A -85,B 0,C 180,E1 17660.72,E2 17660.72} C_VEL
LIN {X 0,Y 478.164,Z 407.035,A -85,B 0,C 180,E1 17658.343,E2 17658.343} C_VEL
LIN {X 0,Y 473.94,Z 401.336,A -85,B 0,C 180,E1 17656.611,E2 17656.611} C_VEL
LIN {X 0,Y 470.717,Z 396.957,A -85,B 0,C 180,E1 17655.146,E2 17655.146} C_VEL
LIN {X 0,Y 466.856,Z 391.882,A -85,B 0,C 180,E1 17653.185,E2 17653.185} C_VEL
LIN {X 0,Y 463.483,Z 387.376,A -85,B 0,C 180,E1 17651.196,E2 17651.196} C_VEL
LIN {X 0,Y 459.417,Z 382.35,A -85,B 0,C 180,E1 17648.259,E2 17648.259} C_VEL
LIN {X 0,Y 458.607,Z 380.965,A -85,B 0,C 180,E1 17647.517,E2 17647.517} C_VEL
LIN {X 0,Y 455.545,Z 377.821,A -85,B 0,C 180,E1 17644.154,E2 17644.154} C_VEL
LIN {X 0,Y 454.553,Z 375.409,A -85,B 0,C 180,E1 17642.143,E2 17642.143} C_VEL
LIN {X 0,Y 453.756,Z 374.846,A -85,B 0,C 180,E1 17637.853,E2 17637.853} C_VEL
LIN {X 0,Y 454.672,Z 375.501,A -85,B 0,C 180,E1 17634.7,E2 17634.7} C_VEL
LIN {X 0,Y 457.019,Z 379.849,A -85,B 0,C 180,E1 17631.064,E2 17631.064} C_VEL
LIN {X 0,Y 459.027,Z 381.468,A -85,B 0,C 180,E1 17629.203,E2 17629.203} C_VEL
LIN {X 0,Y 461.83,Z 385.633,A -85,B 0,C 180,E1 17626.975,E2 17626.975} C_VEL
LIN {X 0,Y 463.493,Z 387.433,A -85,B 0,C 180,E1 17625.891,E2 17625.891} C_VEL
LIN {X 0,Y 466.876,Z 391.9,A -85,B 0,C 180,E1 17623.898,E2 17623.898} C_VEL
LIN {X 0,Y 468.683,Z 394.359,A -85,B 0,C 180,E1 17622.942,E2 17622.942} C_VEL
LIN {X 0,Y 472.134,Z 398.895,A -85,B 0,C 180,E1 17621.286,E2 17621.286} C_VEL
LIN {X 0,Y 476.543,Z 404.92,A -85,B 0,C 180,E1 17619.392,E2 17619.392} C_VEL
LIN {X 0,Y 481.004,Z 411.111,A -85,B 0,C 180,E1 17617.67,E2 17617.67} C_VEL
LIN {X 0,Y 489.438,Z 424.364,A -85,B 0,C 180,E1 17614.757,E2 17614.757} C_VEL
LIN {X 0,Y 496.211,Z 435.771,A -85,B 0,C 180,E1 17612.682,E2 17612.682} C_VEL
LIN {X 0,Y 499.724,Z 442.081,A -85,B 0,C 180,E1 17611.673,E2 17611.673} C_VEL
LIN {X 0,Y 484.848,Z 666.615,A -85,B 0,C 180,E1 17608.155,E2 17608.155} C_VEL
LIN {X 0,Y 481.046,Z 721.802,A -85,B 0,C 180,E1 17607.264,E2 17607.264} C_VEL
LIN {X 0,Y 477.749,Z 748.558,A -85,B 0,C 180,E1 17606.698,E2 17606.698} C_VEL
LIN {X 0,Y 474.19,Z 770.05,A -85,B 0,C 180,E1 17606.113,E2 17606.113} C_VEL
LIN {X 0,Y 469.492,Z 793.829,A -85,B 0,C 180,E1 17605.293,E2 17605.293} C_VEL
LIN {X 0,Y 463.51,Z 818.764,A -85,B 0,C 180,E1 17604.204,E2 17604.204} C_VEL
LIN {X 0,Y 458.084,Z 838.686,A -85,B 0,C 180,E1 17603.153,E2 17603.153} C_VEL
LIN {X 0,Y 451.847,Z 859.377,A -85,B 0,C 180,E1 17601.873,E2 17601.873} C_VEL
LIN {X 0,Y 444.049,Z 882.543,A -85,B 0,C 180,E1 17600.161,E2 17600.161} C_VEL
LIN {X 0,Y 437.396,Z 900.768,A -85,B 0,C 180,E1 17598.574,E2 17598.574} C_VEL
LIN {X 0,Y 430.607,Z 918.339,A -85,B 0,C 180,E1 17596.813,E2 17596.813} C_VEL
LIN {X 0,Y 422.013,Z 939.33,A -85,B 0,C 180,E1 17594.343,E2 17594.343} C_VEL
LIN {X 0,Y 415.095,Z 955.516,A -85,B 0,C 180,E1 17592.105,E2 17592.105} C_VEL
LIN {X 0,Y 408.165,Z 971.487,A -85,B 0,C 180,E1 17589.563,E2 17589.563} C_VEL
LIN {X 0,Y 400.822,Z 988.211,A -85,B 0,C 180,E1 17586.421,E2 17586.421} C_VEL
LIN {X 0,Y 395.327,Z 1000.912,A -85,B 0,C 180,E1 17583.636,E2 17583.636} C_VEL
LIN {X 0,Y 389.915,Z 1013.924,A -85,B 0,C 180,E1 17580.343,E2 17580.343} C_VEL
LIN {X 0,Y 385.172,Z 1025.954,A -85,B 0,C 180,E1 17576.686,E2 17576.686} C_VEL
LIN {X 0,Y 382.104,Z 1034.609,A -85,B 0,C 180,E1 17573.601,E2 17573.601} C_VEL
LIN {X 0,Y 379.323,Z 1043.715,A -85,B 0,C 180,E1 17569.771,E2 17569.771} C_VEL
LIN {X 0,Y 377.521,Z 1050.84,A -85,B 0,C 180,E1 17565.964,E2 17565.964} C_VEL
LIN {X 0,Y 376.614,Z 1055.703,A -85,B 0,C 180,E1 17562.73,E2 17562.73} C_VEL
LIN {X 0,Y 376.129,Z 1059.475,A -85,B 0,C 180,E1 17559.487,E2 17559.487} C_VEL
LIN {X 0,Y 375.929,Z 1062.477,A -85,B 0,C 180,E1 17555.801,E2 17555.801} C_VEL
LIN {X 0,Y 375.908,Z 1063.873,A -85,B 0,C 180,E1 17552.134,E2 17552.134} C_VEL
LIN {X 0,Y 375.913,Z 1063.998,A -85,B 0,C 180,E1 17549.086,E2 17549.086} C_VEL
LIN {X 0,Y 375.913,Z 1063.2,A -85,B 0,C 180,E1 17546.187,E2 17546.187} C_VEL
LIN {X 0,Y 375.972,Z 1061.38,A -85,B 0,C 180,E1 17543.127,E2 17543.127} C_VEL
LIN {X 0,Y 376.167,Z 1058.548,A -85,B 0,C 180,E1 17540.051,E2 17540.051} C_VEL
LIN {X 0,Y 376.797,Z 1053.848,A -85,B 0,C 180,E1 17536.339,E2 17536.339} C_VEL
LIN {X 0,Y 378.028,Z 1047.418,A -85,B 0,C 180,E1 17532.609,E2 17532.609} C_VEL
LIN {X 0,Y 379.77,Z 1040.507,A -85,B 0,C 180,E1 17529.341,E2 17529.341} C_VEL
LIN {X 0,Y 382.436,Z 1031.711,A -85,B 0,C 180,E1 17525.85,E2 17525.85} C_VEL
LIN {X 0,Y 386.387,Z 1020.155,A -85,B 0,C 180,E1 17522.07,E2 17522.07} C_VEL
LIN {X 0,Y 390.424,Z 1009.422,A -85,B 0,C 180,E1 17519.087,E2 17519.087} C_VEL
LIN {X 0,Y 395.741,Z 996.099,A -85,B 0,C 180,E1 17515.881,E2 17515.881} C_VEL
LIN {X 0,Y 401.994,Z 980.622,A -85,B 0,C 180,E1 17512.745,E2 17512.745} C_VEL
LIN {X 0,Y 407.902,Z 966.235,A -85,B 0,C 180,E1 17510.224,E2 17510.224} C_VEL
LIN {X 0,Y 415.232,Z 948.336,A -85,B 0,C 180,E1 17507.511,E2 17507.511} C_VEL
LIN {X 0,Y 422.447,Z 929.852,A -85,B 0,C 180,E1 17505.144,E2 17505.144} C_VEL
LIN {X 0,Y 428.783,Z 913.115,A -85,B 0,C 180,E1 17503.282,E2 17503.282} C_VEL
LIN {X 0,Y 436.327,Z 892.143,A -85,B 0,C 180,E1 17501.267,E2 17501.267} C_VEL
LIN {X 0,Y 443.382,Z 870.637,A -85,B 0,C 180,E1 17499.533,E2 17499.533} C_VEL
LIN {X 0,Y 449.222,Z 851.523,A -85,B 0,C 180,E1 17498.214,E2 17498.214} C_VEL
LIN {X 0,Y 455.839,Z 827.5,A -85,B 0,C 180,E1 17496.81,E2 17496.81} C_VEL
LIN {X 0,Y 460.956,Z 806.113,A -85,B 0,C 180,E1 17495.781,E2 17495.781} C_VEL
LIN {X 0,Y 465.179,Z 786.001,A -85,B 0,C 180,E1 17494.967,E2 17494.967} C_VEL
LIN {X 0,Y 469.747,Z 760.561,A -85,B 0,C 180,E1 17494.133,E2 17494.133} C_VEL
LIN {X 0,Y 473.19,Z 735.088,A -85,B 0,C 180,E1 17493.515,E2 17493.515} C_VEL
LIN {X 0,Y 475.329,Z 712.603,A -85,B 0,C 180,E1 17493.091,E2 17493.091} C_VEL
LIN {X 0,Y 489.534,Z 481.355,A -85,B 0,C 180,E1 17489.444,E2 17489.444} C_VEL
LIN {X 0,Y 492.248,Z 437.546,A -85,B 0,C 180,E1 17488.745,E2 17488.745} C_VEL
LIN {X 0,Y 481.905,Z 419.716,A -85,B 0,C 180,E1 17485.997,E2 17485.997} C_VEL
LIN {X 0,Y 471.792,Z 403.523,A -85,B 0,C 180,E1 17482.952,E2 17482.952} C_VEL
LIN {X 0,Y 463.485,Z 392.333,A -85,B 0,C 180,E1 17480.127,E2 17480.127} C_VEL
LIN {X 0,Y 459.619,Z 387.241,A -85,B 0,C 180,E1 17478.651,E2 17478.651} C_VEL
LIN {X 0,Y 456.159,Z 382.672,A -85,B 0,C 180,E1 17477.213,E2 17477.213} C_VEL
LIN {X 0,Y 452.303,Z 377.69,A -85,B 0,C 180,E1 17475.449,E2 17475.449} C_VEL
LIN {X 0,Y 448.724,Z 372.922,A -85,B 0,C 180,E1 17473.597,E2 17473.597} C_VEL
LIN {X 0,Y 444.799,Z 368.405,A -85,B 0,C 180,E1 17471.278,E2 17471.278} C_VEL
LIN {X 0,Y 443.711,Z 366.71,A -85,B 0,C 180,E1 17470.517,E2 17470.517} C_VEL
LIN {X 0,Y 440.317,Z 363.145,A -85,B 0,C 180,E1 17467.897,E2 17467.897} C_VEL
LIN {X 0,Y 439.145,Z 360.792,A -85,B 0,C 180,E1 17466.668,E2 17466.668} C_VEL
LIN {X 0,Y 435.151,Z 356.737,A -85,B 0,C 180,E1 17459.21,E2 17459.21} C_VEL
LIN {X 0,Y 435.269,Z 356.987,A -85,B 0,C 180,E1 17456.708,E2 17456.708} C_VEL
LIN {X 0,Y 439.377,Z 361.139,A -85,B 0,C 180,E1 17449.908,E2 17449.908} C_VEL
LIN {X 0,Y 441.57,Z 364.839,A -85,B 0,C 180,E1 17447.843,E2 17447.843} C_VEL
LIN {X 0,Y 444.186,Z 367.278,A -85,B 0,C 180,E1 17445.978,E2 17445.978} C_VEL
LIN {X 0,Y 447.232,Z 371.498,A -85,B 0,C 180,E1 17444.038,E2 17444.038} C_VEL
LIN {X 0,Y 448.935,Z 373.28,A -85,B 0,C 180,E1 17443.103,E2 17443.103} C_VEL
LIN {X 0,Y 452.569,Z 377.928,A -85,B 0,C 180,E1 17441.248,E2 17441.248} C_VEL
LIN {X 0,Y 458.1,Z 385.144,A -85,B 0,C 180,E1 17438.79,E2 17438.79} C_VEL
LIN {X 0,Y 462.337,Z 390.738,A -85,B 0,C 180,E1 17437.124,E2 17437.124} C_VEL
LIN {X 0,Y 468.771,Z 399.403,A -85,B 0,C 180,E1 17434.849,E2 17434.849} C_VEL
LIN {X 0,Y 476.344,Z 410.135,A -85,B 0,C 180,E1 17432.463,E2 17432.463} C_VEL
LIN {X 0,Y 484.86,Z 422.851,A -85,B 0,C 180,E1 17430.062,E2 17430.062} C_VEL
LIN {X 0,Y 490.756,Z 432.397,A -85,B 0,C 180,E1 17428.527,E2 17428.527} C_VEL
LIN {X 0,Y 492.327,Z 435.559,A -85,B 0,C 180,E1 17428.118,E2 17428.118} C_VEL
LIN {X 0,Y 479.302,Z 646.05,A -85,B 0,C 180,E1 17424.806,E2 17424.806} C_VEL
LIN {X 0,Y 474.923,Z 715.237,A -85,B 0,C 180,E1 17423.693,E2 17423.693} C_VEL
LIN {X 0,Y 471.74,Z 743.208,A -85,B 0,C 180,E1 17423.092,E2 17423.092} C_VEL
LIN {X 0,Y 468.554,Z 763.911,A -85,B 0,C 180,E1 17422.508,E2 17422.508} C_VEL
LIN {X 0,Y 464.621,Z 785.179,A -85,B 0,C 180,E1 17421.766,E2 17421.766} C_VEL
LIN {X 0,Y 458.73,Z 811.93,A -85,B 0,C 180,E1 17420.597,E2 17420.597} C_VEL
LIN {X 0,Y 453.54,Z 832.168,A -85,B 0,C 180,E1 17419.516,E2 17419.516} C_VEL
LIN {X 0,Y 447.993,Z 851.728,A -85,B 0,C 180,E1 17418.295,E2 17418.295} C_VEL
LIN {X 0,Y 440.642,Z 875.169,A -85,B 0,C 180,E1 17416.563,E2 17416.563} C_VEL
LIN {X 0,Y 433.882,Z 894.754,A -85,B 0,C 180,E1 17414.844,E2 17414.844} C_VEL
LIN {X 0,Y 427.282,Z 912.831,A -85,B 0,C 180,E1 17413.011,E2 17413.011} C_VEL
LIN {X 0,Y 419.223,Z 933.613,A -85,B 0,C 180,E1 17410.537,E2 17410.537} C_VEL
LIN {X 0,Y 412.799,Z 949.5,A -85,B 0,C 180,E1 17408.322,E2 17408.322} C_VEL
LIN {X 0,Y 406.43,Z 965.023,A -85,B 0,C 180,E1 17405.84,E2 17405.84} C_VEL
LIN {X 0,Y 399.522,Z 981.626,A -85,B 0,C 180,E1 17402.723,E2 17402.723} C_VEL
LIN {X 0,Y 394.334,Z 994.211,A -85,B 0,C 180,E1 17399.968,E2 17399.968} C_VEL
LIN {X 0,Y 389.258,Z 1007.089,A -85,B 0,C 180,E1 17396.713,E2 17396.713} C_VEL
LIN {X 0,Y 384.739,Z 1019.1,A -85,B 0,C 180,E1 17393.073,E2 17393.073} C_VEL
LIN {X 0,Y 381.743,Z 1027.958,A -85,B 0,C 180,E1 17389.908,E2 17389.908} C_VEL
LIN {X 0,Y 379.113,Z 1036.984,A -85,B 0,C 180,E1 17386.077,E2 17386.077} C_VEL
LIN {X 0,Y 377.47,Z 1043.824,A -85,B 0,C 180,E1 17382.39,E2 17382.39} C_VEL
LIN {X 0,Y 376.637,Z 1048.418,A -85,B 0,C 180,E1 17379.319,E2 17379.319} C_VEL
LIN {X 0,Y 376.153,Z 1052.149,A -85,B 0,C 180,E1 17376.104,E2 17376.104} C_VEL
LIN {X 0,Y 375.948,Z 1055.132,A -85,B 0,C 180,E1 17372.439,E2 17372.439} C_VEL
LIN {X 0,Y 375.908,Z 1056.55,A -85,B 0,C 180,E1 17368.781,E2 17368.781} C_VEL
LIN {X 0,Y 375.908,Z 1056.701,A -85,B 0,C 180,E1 17365.729,E2 17365.729} C_VEL
LIN {X 0,Y 375.935,Z 1055.93,A -85,B 0,C 180,E1 17362.789,E2 17362.789} C_VEL
LIN {X 0,Y 376.034,Z 1054.145,A -85,B 0,C 180,E1 17359.689,E2 17359.689} C_VEL
LIN {X 0,Y 376.323,Z 1051.257,A -85,B 0,C 180,E1 17356.478,E2 17356.478} C_VEL
LIN {X 0,Y 377.181,Z 1046.34,A -85,B 0,C 180,E1 17352.569,E2 17352.569} C_VEL
LIN {X 0,Y 377.243,Z 1046.031,A -85,B 0,C 180,E1 17352.379,E2 17352.379} C_VEL
LIN {X 0,Y 376.651,Z 1044.298,A -85,B 0,C 180,E1 17351.235,E2 17351.235} C_VEL
LIN {X 0,Y 371.709,Z 1039.337,A -85,B 0,C 180,E1 17348.066,E2 17348.066} C_VEL
LIN {X 0,Y 371.612,Z 1037.666,A -85,B 0,C 180,E1 17347.155,E2 17347.155} C_VEL
LIN {X 0,Y 374.61,Z 1028.78,A -85,B 0,C 180,E1 17343.187,E2 17343.187} C_VEL
LIN {X 0,Y 378.035,Z 1019.85,A -85,B 0,C 180,E1 17339.872,E2 17339.872} C_VEL
LIN {X 0,Y 382.975,Z 1008.259,A -85,B 0,C 180,E1 17336.213,E2 17336.213} C_VEL
LIN {X 0,Y 388.759,Z 995.241,A -85,B 0,C 180,E1 17332.813,E2 17332.813} C_VEL
LIN {X 0,Y 394.298,Z 983.176,A -85,B 0,C 180,E1 17330.091,E2 17330.091} C_VEL
LIN {X 0,Y 401.698,Z 967.313,A -85,B 0,C 180,E1 17326.998,E2 17326.998} C_VEL
LIN {X 0,Y 409.456,Z 950.204,A -85,B 0,C 180,E1 17324.212,E2 17324.212} C_VEL
LIN {X 0,Y 416.449,Z 934.525,A -85,B 0,C 180,E1 17322.004,E2 17322.004} C_VEL
LIN {X 0,Y 425.241,Z 913.985,A -85,B 0,C 180,E1 17319.535,E2 17319.535} C_VEL
LIN {X 0,Y 432.608,Z 895.561,A -85,B 0,C 180,E1 17317.663,E2 17317.663} C_VEL
LIN {X 0,Y 439.491,Z 877.271,A -85,B 0,C 180,E1 17316.055,E2 17316.055} C_VEL
LIN {X 0,Y 447.734,Z 853.372,A -85,B 0,C 180,E1 17314.281,E2 17314.281} C_VEL
LIN {X 0,Y 453.869,Z 833.48,A -85,B 0,C 180,E1 17313.044,E2 17313.044} C_VEL
LIN {X 0,Y 459.593,Z 812.88,A -85,B 0,C 180,E1 17311.953,E2 17311.953} C_VEL
LIN {X 0,Y 465.952,Z 786.379,A -85,B 0,C 180,E1 17310.807,E2 17310.807} C_VEL
LIN {X 0,Y 470.414,Z 763.953,A -85,B 0,C 180,E1 17310.038,E2 17310.038} C_VEL
LIN {X 0,Y 473.933,Z 742.685,A -85,B 0,C 180,E1 17309.456,E2 17309.456} C_VEL
LIN {X 0,Y 477.327,Z 714.486,A -85,B 0,C 180,E1 17308.867,E2 17308.867} C_VEL
LIN {X 0,Y 483.781,Z 620.543,A -85,B 0,C 180,E1 17307.371,E2 17307.371} C_VEL
LIN {X 0,Y 495.84,Z 444.001,A -85,B 0,C 180,E1 17304.593,E2 17304.593} C_VEL
LIN {X 0,Y 490.286,Z 434.837,A -85,B 0,C 180,E1 17302.925,E2 17302.925} C_VEL
LIN {X 0,Y 482.056,Z 422.584,A -85,B 0,C 180,E1 17300.204,E2 17300.204} C_VEL
LIN {X 0,Y 475.855,Z 413.835,A -85,B 0,C 180,E1 17297.866,E2 17297.866} C_VEL
LIN {X 0,Y 472.013,Z 408.528,A -85,B 0,C 180,E1 17296.238,E2 17296.238} C_VEL
LIN {X 0,Y 468.985,Z 404.361,A -85,B 0,C 180,E1 17294.824,E2 17294.824} C_VEL
LIN {X 0,Y 465.32,Z 399.459,A -85,B 0,C 180,E1 17292.913,E2 17292.913} C_VEL
LIN {X 0,Y 461.566,Z 394.356,A -85,B 0,C 180,E1 17290.611,E2 17290.611} C_VEL
LIN {X 0,Y 458.282,Z 390.297,A -85,B 0,C 180,E1 17288.153,E2 17288.153} C_VEL
LIN {X 0,Y 457.492,Z 388.845,A -85,B 0,C 180,E1 17287.409,E2 17287.409} C_VEL
LIN {X 0,Y 454.483,Z 385.696,A -85,B 0,C 180,E1 17284.037,E2 17284.037} C_VEL
LIN {X 0,Y 453.521,Z 383.307,A -85,B 0,C 180,E1 17282.022,E2 17282.022} C_VEL
LIN {X 0,Y 452.794,Z 382.792,A -85,B 0,C 180,E1 17277.722,E2 17277.722} C_VEL
LIN {X 0,Y 453.683,Z 383.584,A -85,B 0,C 180,E1 17274.689,E2 17274.689} C_VEL
LIN {X 0,Y 456.049,Z 387.84,A -85,B 0,C 180,E1 17271.044,E2 17271.044} C_VEL
LIN {X 0,Y 457.895,Z 389.435,A -85,B 0,C 180,E1 17269.31,E2 17269.31} C_VEL
LIN {X 0,Y 460.892,Z 393.739,A -85,B 0,C 180,E1 17266.928,E2 17266.928} C_VEL
LIN {X 0,Y 462.225,Z 395.315,A -85,B 0,C 180,E1 17266.043,E2 17266.043} C_VEL
LIN {X 0,Y 465.689,Z 399.812,A -85,B 0,C 180,E1 17263.984,E2 17263.984} C_VEL
LIN {X 0,Y 470.513,Z 406.46,A -85,B 0,C 180,E1 17261.54,E2 17261.54} C_VEL
LIN {X 0,Y 475.063,Z 412.792,A -85,B 0,C 180,E1 17259.55,E2 17259.55} C_VEL
LIN {X 0,Y 479.088,Z 418.495,A -85,B 0,C 180,E1 17257.966,E2 17257.966} C_VEL
LIN {X 0,Y 487.229,Z 431.538,A -85,B 0,C 180,E1 17255.089,E2 17255.089} C_VEL
LIN {X 0,Y 493.802,Z 442.834,A -85,B 0,C 180,E1 17253.027,E2 17253.027} C_VEL
LIN {X 0,Y 495.81,Z 446.528,A -85,B 0,C 180,E1 17252.43,E2 17252.43} C_VEL
LIN {X 0,Y 480.369,Z 673.387,A -85,B 0,C 180,E1 17248.872,E2 17248.872} C_VEL
LIN {X 0,Y 476.804,Z 723.002,A -85,B 0,C 180,E1 17248.065,E2 17248.065} C_VEL
LIN {X 0,Y 473.44,Z 749.128,A -85,B 0,C 180,E1 17247.508,E2 17247.508} C_VEL
LIN {X 0,Y 469.802,Z 770.512,A -85,B 0,C 180,E1 17246.925,E2 17246.925} C_VEL
LIN {X 0,Y 464.675,Z 795.742,A -85,B 0,C 180,E1 17246.049,E2 17246.049} C_VEL
LIN {X 0,Y 458.854,Z 819.11,A -85,B 0,C 180,E1 17245.019,E2 17245.019} C_VEL
LIN {X 0,Y 453.191,Z 839.334,A -85,B 0,C 180,E1 17243.949,E2 17243.949} C_VEL
LIN {X 0,Y 446.34,Z 861.4,A -85,B 0,C 180,E1 17242.575,E2 17242.575} C_VEL
LIN {X 0,Y 438.608,Z 883.468,A -85,B 0,C 180,E1 17240.917,E2 17240.917} C_VEL
LIN {X 0,Y 432.033,Z 900.938,A -85,B 0,C 180,E1 17239.386,E2 17239.386} C_VEL
LIN {X 0,Y 424.903,Z 918.815,A -85,B 0,C 180,E1 17237.584,E2 17237.584} C_VEL
LIN {X 0,Y 415.935,Z 939.942,A -85,B 0,C 180,E1 17235.069,E2 17235.069} C_VEL
LIN {X 0,Y 409.275,Z 955.005,A -85,B 0,C 180,E1 17232.97,E2 17232.97} C_VEL
LIN {X 0,Y 402.56,Z 969.879,A -85,B 0,C 180,E1 17230.599,E2 17230.599} C_VEL
LIN {X 0,Y 394.383,Z 987.772,A -85,B 0,C 180,E1 17227.241,E2 17227.241} C_VEL
LIN {X 0,Y 388.702,Z 1000.313,A -85,B 0,C 180,E1 17224.466,E2 17224.466} C_VEL
LIN {X 0,Y 383.23,Z 1012.802,A -85,B 0,C 180,E1 17221.279,E2 17221.279} C_VEL
LIN {X 0,Y 377.96,Z 1025.496,A -85,B 0,C 180,E1 17217.407,E2 17217.407} C_VEL
LIN {X 0,Y 374.663,Z 1034.194,A -85,B 0,C 180,E1 17214.267,E2 17214.267} C_VEL
LIN {X 0,Y 371.937,Z 1042.4,A -85,B 0,C 180,E1 17210.785,E2 17210.785} C_VEL
LIN {X 0,Y 369.784,Z 1050.252,A -85,B 0,C 180,E1 17206.656,E2 17206.656} C_VEL
LIN {X 0,Y 368.74,Z 1055.242,A -85,B 0,C 180,E1 17203.326,E2 17203.326} C_VEL
LIN {X 0,Y 368.196,Z 1058.94,A -85,B 0,C 180,E1 17200.167,E2 17200.167} C_VEL
LIN {X 0,Y 367.972,Z 1061.739,A -85,B 0,C 180,E1 17196.867,E2 17196.867} C_VEL
LIN {X 0,Y 367.913,Z 1063.682,A -85,B 0,C 180,E1 17192.96,E2 17192.96} C_VEL
LIN {X 0,Y 367.912,Z 1063.962,A -85,B 0,C 180,E1 17189.377,E2 17189.377} C_VEL
LIN {X 0,Y 367.912,Z 1063.179,A -85,B 0,C 180,E1 17186.26,E2 17186.26} C_VEL
LIN {X 0,Y 367.971,Z 1061.398,A -85,B 0,C 180,E1 17183.133,E2 17183.133} C_VEL
LIN {X 0,Y 368.173,Z 1058.605,A -85,B 0,C 180,E1 17179.991,E2 17179.991} C_VEL
LIN {X 0,Y 368.752,Z 1054.361,A -85,B 0,C 180,E1 17176.515,E2 17176.515} C_VEL
LIN {X 0,Y 370.119,Z 1047.593,A -85,B 0,C 180,E1 17172.388,E2 17172.388} C_VEL
LIN {X 0,Y 371.94,Z 1040.724,A -85,B 0,C 180,E1 17169.051,E2 17169.051} C_VEL
LIN {X 0,Y 374.51,Z 1032.578,A -85,B 0,C 180,E1 17165.723,E2 17165.723} C_VEL
LIN {X 0,Y 378.848,Z 1020.503,A -85,B 0,C 180,E1 17161.636,E2 17161.636} C_VEL
LIN {X 0,Y 383.142,Z 1009.583,A -85,B 0,C 180,E1 17158.538,E2 17158.538} C_VEL
LIN {X 0,Y 388.558,Z 996.545,A -85,B 0,C 180,E1 17155.34,E2 17155.34} C_VEL
LIN {X 0,Y 395.251,Z 980.698,A -85,B 0,C 180,E1 17152.068,E2 17152.068} C_VEL
LIN {X 0,Y 401.155,Z 966.853,A -85,B 0,C 180,E1 17149.605,E2 17149.605} C_VEL
LIN {X 0,Y 408.718,Z 949.079,A -85,B 0,C 180,E1 17146.861,E2 17146.861} C_VEL
LIN {X 0,Y 416.37,Z 930.125,A -85,B 0,C 180,E1 17144.404,E2 17144.404} C_VEL
LIN {X 0,Y 422.777,Z 913.745,A -85,B 0,C 180,E1 17142.564,E2 17142.564} C_VEL
LIN {X 0,Y 430.42,Z 893.257,A -85,B 0,C 180,E1 17140.568,E2 17140.568} C_VEL
LIN {X 0,Y 437.655,Z 871.891,A -85,B 0,C 180,E1 17138.825,E2 17138.825} C_VEL
LIN {X 0,Y 443.636,Z 852.924,A -85,B 0,C 180,E1 17137.5,E2 17137.5} C_VEL
LIN {X 0,Y 450.133,Z 830.346,A -85,B 0,C 180,E1 17136.153,E2 17136.153} C_VEL
LIN {X 0,Y 455.94,Z 806.847,A -85,B 0,C 180,E1 17135.006,E2 17135.006} C_VEL
LIN {X 0,Y 460.269,Z 786.819,A -85,B 0,C 180,E1 17134.192,E2 17134.192} C_VEL
LIN {X 0,Y 464.587,Z 763.477,A -85,B 0,C 180,E1 17133.414,E2 17133.414} C_VEL
LIN {X 0,Y 468.456,Z 736.648,A -85,B 0,C 180,E1 17132.744,E2 17132.744} C_VEL
LIN {X 0,Y 470.697,Z 714.257,A -85,B 0,C 180,E1 17132.315,E2 17132.315} C_VEL
LIN {X 0,Y 485.265,Z 484.482,A -85,B 0,C 180,E1 17128.68,E2 17128.68} C_VEL
LIN {X 0,Y 487.95,Z 441.704,A -85,B 0,C 180,E1 17127.986,E2 17127.986} C_VEL
LIN {X 0,Y 478.455,Z 425.114,A -85,B 0,C 180,E1 17125.367,E2 17125.367} C_VEL
LIN {X 0,Y 469.191,Z 410.202,A -85,B 0,C 180,E1 17122.491,E2 17122.491} C_VEL
LIN {X 0,Y 461.46,Z 399.582,A -85,B 0,C 180,E1 17119.789,E2 17119.789} C_VEL
LIN {X 0,Y 457.588,Z 394.41,A -85,B 0,C 180,E1 17118.274,E2 17118.274} C_VEL
LIN {X 0,Y 454.337,Z 390.053,A -85,B 0,C 180,E1 17116.888,E2 17116.888} C_VEL
LIN {X 0,Y 450.685,Z 385.245,A -85,B 0,C 180,E1 17115.177,E2 17115.177} C_VEL
LIN {X 0,Y 446.72,Z 380.023,A -85,B 0,C 180,E1 17113.066,E2 17113.066} C_VEL
LIN {X 0,Y 443.343,Z 375.94,A -85,B 0,C 180,E1 17110.986,E2 17110.986} C_VEL
LIN {X 0,Y 442.36,Z 374.462,A -85,B 0,C 180,E1 17110.286,E2 17110.286} C_VEL
LIN {X 0,Y 439.058,Z 370.829,A -85,B 0,C 180,E1 17107.656,E2 17107.656} C_VEL
LIN {X 0,Y 437.909,Z 368.617,A -85,B 0,C 180,E1 17106.424,E2 17106.424} C_VEL
LIN {X 0,Y 434.175,Z 364.68,A -85,B 0,C 180,E1 17099.208,E2 17099.208} C_VEL
LIN {X 0,Y 434.293,Z 364.946,A -85,B 0,C 180,E1 17096.7,E2 17096.7} C_VEL
LIN {X 0,Y 438.208,Z 368.986,A -85,B 0,C 180,E1 17090.08,E2 17090.08} C_VEL
LIN {X 0,Y 440.441,Z 372.731,A -85,B 0,C 180,E1 17087.944,E2 17087.944} C_VEL
LIN {X 0,Y 442.901,Z 375.124,A -85,B 0,C 180,E1 17086.154,E2 17086.154} C_VEL
LIN {X 0,Y 446.051,Z 379.41,A -85,B 0,C 180,E1 17084.128,E2 17084.128} C_VEL
LIN {X 0,Y 447.501,Z 381.028,A -85,B 0,C 180,E1 17083.314,E2 17083.314} C_VEL
LIN {X 0,Y 452.093,Z 387.123,A -85,B 0,C 180,E1 17080.96,E2 17080.96} C_VEL
LIN {X 0,Y 456.471,Z 392.826,A -85,B 0,C 180,E1 17079.014,E2 17079.014} C_VEL
LIN {X 0,Y 460.654,Z 398.44,A -85,B 0,C 180,E1 17077.339,E2 17077.339} C_VEL
LIN {X 0,Y 466.842,Z 406.949,A -85,B 0,C 180,E1 17075.111,E2 17075.111} C_VEL
LIN {X 0,Y 473.862,Z 417.026,A -85,B 0,C 180,E1 17072.851,E2 17072.851} C_VEL
LIN {X 0,Y 482.244,Z 429.751,A -85,B 0,C 180,E1 17070.431,E2 17070.431} C_VEL
LIN {X 0,Y 487.89,Z 439.088,A -85,B 0,C 180,E1 17068.924,E2 17068.924} C_VEL
LIN {X 0,Y 488.052,Z 440.077,A -85,B 0,C 180,E1 17068.861,E2 17068.861} C_VEL
LIN {X 0,Y 474.436,Z 654.047,A -85,B 0,C 180,E1 17065.487,E2 17065.487} C_VEL
LIN {X 0,Y 470.373,Z 715.866,A -85,B 0,C 180,E1 17064.487,E2 17064.487} C_VEL
LIN {X 0,Y 467.149,Z 743.365,A -85,B 0,C 180,E1 17063.894,E2 17063.894} C_VEL
LIN {X 0,Y 463.887,Z 764.05,A -85,B 0,C 180,E1 17063.312,E2 17063.312} C_VEL
LIN {X 0,Y 459.734,Z 785.958,A -85,B 0,C 180,E1 17062.546,E2 17062.546} C_VEL
LIN {X 0,Y 453.696,Z 812.55,A -85,B 0,C 180,E1 17061.377,E2 17061.377} C_VEL
LIN {X 0,Y 448.204,Z 833.363,A -85,B 0,C 180,E1 17060.258,E2 17060.258} C_VEL
LIN {X 0,Y 441.709,Z 855.533,A -85,B 0,C 180,E1 17058.851,E2 17058.851} C_VEL
LIN {X 0,Y 434.367,Z 877.78,A -85,B 0,C 180,E1 17057.152,E2 17057.152} C_VEL
LIN {X 0,Y 427.944,Z 895.818,A -85,B 0,C 180,E1 17055.544,E2 17055.544} C_VEL
LIN {X 0,Y 420.506,Z 915.55,A -85,B 0,C 180,E1 17053.511,E2 17053.511} C_VEL
LIN {X 0,Y 412.649,Z 934.944,A -85,B 0,C 180,E1 17051.137,E2 17051.137} C_VEL
LIN {X 0,Y 406.044,Z 950.723,A -85,B 0,C 180,E1 17048.898,E2 17048.898} C_VEL
LIN {X 0,Y 398.808,Z 967.78,A -85,B 0,C 180,E1 17046.099,E2 17046.099} C_VEL
LIN {X 0,Y 392.05,Z 983.265,A -85,B 0,C 180,E1 17043.078,E2 17043.078} C_VEL
LIN {X 0,Y 386.732,Z 995.704,A -85,B 0,C 180,E1 17040.276,E2 17040.276} C_VEL
LIN {X 0,Y 381.096,Z 1009.412,A -85,B 0,C 180,E1 17036.657,E2 17036.657} C_VEL
LIN {X 0,Y 376.921,Z 1020.111,A -85,B 0,C 180,E1 17033.282,E2 17033.282} C_VEL
LIN {X 0,Y 373.69,Z 1029.34,A -85,B 0,C 180,E1 17029.866,E2 17029.866} C_VEL
LIN {X 0,Y 370.948,Z 1038.365,A -85,B 0,C 180,E1 17025.783,E2 17025.783} C_VEL
LIN {X 0,Y 369.51,Z 1044.22,A -85,B 0,C 180,E1 17022.502,E2 17022.502} C_VEL
LIN {X 0,Y 368.613,Z 1048.958,A -85,B 0,C 180,E1 17019.209,E2 17019.209} C_VEL
LIN {X 0,Y 368.108,Z 1053.058,A -85,B 0,C 180,E1 17015.455,E2 17015.455} C_VEL
LIN {X 0,Y 367.926,Z 1055.658,A -85,B 0,C 180,E1 17011.557,E2 17011.557} C_VEL
LIN {X 0,Y 367.905,Z 1056.678,A -85,B 0,C 180,E1 17008.443,E2 17008.443} C_VEL
LIN {X 0,Y 367.908,Z 1056.75,A -85,B 0,C 180,E1 17005.479,E2 17005.479} C_VEL
LIN {X 0,Y 367.93,Z 1055.937,A -85,B 0,C 180,E1 17002.505,E2 17002.505} C_VEL
LIN {X 0,Y 368.058,Z 1054.116,A -85,B 0,C 180,E1 16999.354,E2 16999.354} C_VEL
LIN {X 0,Y 368.429,Z 1050.976,A -85,B 0,C 180,E1 16995.862,E2 16995.862} C_VEL
LIN {X 0,Y 369.479,Z 1045.59,A -85,B 0,C 180,E1 16991.704,E2 16991.704} C_VEL
LIN {X 0,Y 371.028,Z 1039.574,A -85,B 0,C 180,E1 16988.167,E2 16988.167} C_VEL
LIN {X 0,Y 371.612,Z 1037.666,A -85,B 0,C 180,E1 16987.155,E2 16987.155} C_VEL
LIN {X 0,Y 371.383,Z 1035.512,A -85,B 0,C 180,E1 16986.006,E2 16986.006} C_VEL
LIN {X 0,Y 367.586,Z 1029.392,A -85,B 0,C 180,E1 16982.902,E2 16982.902} C_VEL
LIN {X 0,Y 367.77,Z 1027.089,A -85,B 0,C 180,E1 16981.925,E2 16981.925} C_VEL
LIN {X 0,Y 372.22,Z 1016.581,A -85,B 0,C 180,E1 16978.089,E2 16978.089} C_VEL
LIN {X 0,Y 377.531,Z 1004.759,A -85,B 0,C 180,E1 16974.548,E2 16974.548} C_VEL
LIN {X 0,Y 382.964,Z 993.24,A -85,B 0,C 180,E1 16971.582,E2 16971.582} C_VEL
LIN {X 0,Y 389.957,Z 978.843,A -85,B 0,C 180,E1 16968.387,E2 16968.387} C_VEL
LIN {X 0,Y 397.556,Z 962.919,A -85,B 0,C 180,E1 16965.436,E2 16965.436} C_VEL
LIN {X 0,Y 404.52,Z 948.201,A -85,B 0,C 180,E1 16963.079,E2 16963.079} C_VEL
LIN {X 0,Y 413.053,Z 929.7,A -85,B 0,C 180,E1 16960.526,E2 16960.526} C_VEL
LIN {X 0,Y 421.25,Z 910.69,A -85,B 0,C 180,E1 16958.327,E2 16958.327} C_VEL
LIN {X 0,Y 428.03,Z 894.187,A -85,B 0,C 180,E1 16956.676,E2 16956.676} C_VEL
LIN {X 0,Y 435.904,Z 873.799,A -85,B 0,C 180,E1 16954.911,E2 16954.911} C_VEL
LIN {X 0,Y 443.398,Z 852.231,A -85,B 0,C 180,E1 16953.349,E2 16953.349} C_VEL
LIN {X 0,Y 449.442,Z 833.07,A -85,B 0,C 180,E1 16952.166,E2 16952.166} C_VEL
LIN {X 0,Y 455.398,Z 812.091,A -85,B 0,C 180,E1 16951.063,E2 16951.063} C_VEL
LIN {X 0,Y 461.82,Z 785.745,A -85,B 0,C 180,E1 16949.936,E2 16949.936} C_VEL
LIN {X 0,Y 466.283,Z 763.749,A -85,B 0,C 180,E1 16949.188,E2 16949.188} C_VEL
LIN {X 0,Y 470.016,Z 741.599,A -85,B 0,C 180,E1 16948.588,E2 16948.588} C_VEL
LIN {X 0,Y 473.35,Z 714.016,A -85,B 0,C 180,E1 16948.022,E2 16948.022} C_VEL
LIN {X 0,Y 482.09,Z 589.471,A -85,B 0,C 180,E1 16946.044,E2 16946.044} C_VEL
LIN {X 0,Y 492.023,Z 448.532,A -85,B 0,C 180,E1 16943.826,E2 16943.826} C_VEL
LIN {X 0,Y 486.221,Z 439.235,A -85,B 0,C 180,E1 16942.011,E2 16942.011} C_VEL
LIN {X 0,Y 478.264,Z 427.116,A -85,B 0,C 180,E1 16939.225,E2 16939.225} C_VEL
LIN {X 0,Y 471.159,Z 417.067,A -85,B 0,C 180,E1 16936.331,E2 16936.331} C_VEL
LIN {X 0,Y 467.269,Z 411.76,A -85,B 0,C 180,E1 16934.499,E2 16934.499} C_VEL
LIN {X 0,Y 463.904,Z 407.145,A -85,B 0,C 180,E1 16932.7,E2 16932.7} C_VEL
LIN {X 0,Y 460.033,Z 401.91,A -85,B 0,C 180,E1 16930.267,E2 16930.267} C_VEL
LIN {X 0,Y 456.951,Z 397.847,A -85,B 0,C 180,E1 16927.861,E2 16927.861} C_VEL
LIN {X 0,Y 456.237,Z 396.631,A -85,B 0,C 180,E1 16927.176,E2 16927.176} C_VEL
LIN {X 0,Y 453.273,Z 393.291,A -85,B 0,C 180,E1 16923.668,E2 16923.668} C_VEL
LIN {X 0,Y 452.492,Z 391.205,A -85,B 0,C 180,E1 16921.9,E2 16921.9} C_VEL
LIN {X 0,Y 451.833,Z 390.744,A -85,B 0,C 180,E1 16917.59,E2 16917.59} C_VEL
LIN {X 0,Y 452.65,Z 391.48,A -85,B 0,C 180,E1 16914.804,E2 16914.804} C_VEL
LIN {X 0,Y 454.963,Z 395.72,A -85,B 0,C 180,E1 16911.15,E2 16911.15} C_VEL
LIN {X 0,Y 456.715,Z 397.286,A -85,B 0,C 180,E1 16909.467,E2 16909.467} C_VEL
LIN {X 0,Y 459.7,Z 401.587,A -85,B 0,C 180,E1 16907.054,E2 16907.054} C_VEL
LIN {X 0,Y 460.962,Z 403.184,A -85,B 0,C 180,E1 16906.196,E2 16906.196} C_VEL
LIN {X 0,Y 465.141,Z 408.772,A -85,B 0,C 180,E1 16903.708,E2 16903.708} C_VEL
LIN {X 0,Y 469.024,Z 414.215,A -85,B 0,C 180,E1 16901.737,E2 16901.737} C_VEL
LIN {X 0,Y 473.518,Z 420.552,A -85,B 0,C 180,E1 16899.738,E2 16899.738} C_VEL
LIN {X 0,Y 477.488,Z 426.366,A -85,B 0,C 180,E1 16898.147,E2 16898.147} C_VEL
LIN {X 0,Y 485.12,Z 438.852,A -85,B 0,C 180,E1 16895.396,E2 16895.396} C_VEL
LIN {X 0,Y 491.591,Z 450.211,A -85,B 0,C 180,E1 16893.32,E2 16893.32} C_VEL
LIN {X 0,Y 491.965,Z 451.212,A -85,B 0,C 180,E1 16893.195,E2 16893.195} C_VEL
LIN {X 0,Y 475.922,Z 680.856,A -85,B 0,C 180,E1 16889.591,E2 16889.591} C_VEL
LIN {X 0,Y 472.618,Z 724.579,A -85,B 0,C 180,E1 16888.874,E2 16888.874} C_VEL
LIN {X 0,Y 469.188,Z 749.969,A -85,B 0,C 180,E1 16888.325,E2 16888.325} C_VEL
LIN {X 0,Y 465.433,Z 771.413,A -85,B 0,C 180,E1 16887.738,E2 16887.738} C_VEL
LIN {X 0,Y 460.247,Z 796.158,A -85,B 0,C 180,E1 16886.877,E2 16886.877} C_VEL
LIN {X 0,Y 454.292,Z 819.456,A -85,B 0,C 180,E1 16885.849,E2 16885.849} C_VEL
LIN {X 0,Y 448.609,Z 839.254,A -85,B 0,C 180,E1 16884.804,E2 16884.804} C_VEL
LIN {X 0,Y 441.747,Z 860.792,A -85,B 0,C 180,E1 16883.466,E2 16883.466} C_VEL
LIN {X 0,Y 433.802,Z 882.937,A -85,B 0,C 180,E1 16881.812,E2 16881.812} C_VEL
LIN {X 0,Y 426.892,Z 900.778,A -85,B 0,C 180,E1 16880.25,E2 16880.25} C_VEL
LIN {X 0,Y 419.298,Z 919.241,A -85,B 0,C 180,E1 16878.382,E2 16878.382} C_VEL
LIN {X 0,Y 410.393,Z 939.549,A -85,B 0,C 180,E1 16875.951,E2 16875.951} C_VEL
LIN {X 0,Y 403.267,Z 955.098,A -85,B 0,C 180,E1 16873.77,E2 16873.77} C_VEL
LIN {X 0,Y 396.306,Z 969.955,A -85,B 0,C 180,E1 16871.378,E2 16871.378} C_VEL
LIN {X 0,Y 387.899,Z 987.609,A -85,B 0,C 180,E1 16868.03,E2 16868.03} C_VEL
LIN {X 0,Y 381.865,Z 1000.349,A -85,B 0,C 180,E1 16865.173,E2 16865.173} C_VEL
LIN {X 0,Y 376.146,Z 1012.825,A -85,B 0,C 180,E1 16861.937,E2 16861.937} C_VEL
LIN {X 0,Y 370.755,Z 1025.125,A -85,B 0,C 180,E1 16858.129,E2 16858.129} C_VEL
LIN {X 0,Y 367.121,Z 1034.185,A -85,B 0,C 180,E1 16854.799,E2 16854.799} C_VEL
LIN {X 0,Y 364.23,Z 1042.382,A -85,B 0,C 180,E1 16851.246,E2 16851.246} C_VEL
LIN {X 0,Y 361.928,Z 1050.216,A -85,B 0,C 180,E1 16847.028,E2 16847.028} C_VEL
LIN {X 0,Y 360.81,Z 1055.198,A -85,B 0,C 180,E1 16843.624,E2 16843.624} C_VEL
LIN {X 0,Y 360.221,Z 1058.888,A -85,B 0,C 180,E1 16840.395,E2 16840.395} C_VEL
LIN {X 0,Y 359.978,Z 1061.679,A -85,B 0,C 180,E1 16837.02,E2 16837.02} C_VEL
LIN {X 0,Y 359.913,Z 1063.608,A -85,B 0,C 180,E1 16833.026,E2 16833.026} C_VEL
LIN {X 0,Y 359.912,Z 1063.88,A -85,B 0,C 180,E1 16829.363,E2 16829.363} C_VEL
LIN {X 0,Y 359.913,Z 1063.09,A -85,B 0,C 180,E1 16826.177,E2 16826.177} C_VEL
LIN {X 0,Y 359.978,Z 1061.301,A -85,B 0,C 180,E1 16822.98,E2 16822.98} C_VEL
LIN {X 0,Y 360.193,Z 1058.5,A -85,B 0,C 180,E1 16819.766,E2 16819.766} C_VEL
LIN {X 0,Y 360.863,Z 1054.038,A -85,B 0,C 180,E1 16816.051,E2 16816.051} C_VEL
LIN {X 0,Y 362.292,Z 1047.461,A -85,B 0,C 180,E1 16811.995,E2 16811.995} C_VEL
LIN {X 0,Y 364.28,Z 1040.423,A -85,B 0,C 180,E1 16808.514,E2 16808.514} C_VEL
LIN {X 0,Y 367.107,Z 1032.015,A -85,B 0,C 180,E1 16805.028,E2 16805.028} C_VEL
LIN {X 0,Y 371.564,Z 1020.236,A -85,B 0,C 180,E1 16800.996,E2 16800.996} C_VEL
LIN {X 0,Y 376.039,Z 1009.397,A -85,B 0,C 180,E1 16797.873,E2 16797.873} C_VEL
LIN {X 0,Y 381.707,Z 996.347,A -85,B 0,C 180,E1 16794.626,E2 16794.626} C_VEL
LIN {X 0,Y 388.695,Z 980.473,A -85,B 0,C 180,E1 16791.311,E2 16791.311} C_VEL
LIN {X 0,Y 394.837,Z 966.614,A -85,B 0,C 180,E1 16788.82,E2 16788.82} C_VEL
LIN {X 0,Y 402.6,Z 948.988,A -85,B 0,C 180,E1 16786.075,E2 16786.075} C_VEL
LIN {X 0,Y 410.364,Z 930.396,A -85,B 0,C 180,E1 16783.642,E2 16783.642} C_VEL
LIN {X 0,Y 417.247,Z 913.339,A -85,B 0,C 180,E1 16781.714,E2 16781.714} C_VEL
LIN {X 0,Y 425.344,Z 892.168,A -85,B 0,C 180,E1 16779.657,E2 16779.657} C_VEL
LIN {X 0,Y 432.774,Z 870.785,A -85,B 0,C 180,E1 16777.921,E2 16777.921} C_VEL
LIN {X 0,Y 439.01,Z 851.455,A -85,B 0,C 180,E1 16776.581,E2 16776.581} C_VEL
LIN {X 0,Y 445.905,Z 827.729,A -85,B 0,C 180,E1 16775.19,E2 16775.19} C_VEL
LIN {X 0,Y 451.312,Z 806.277,A -85,B 0,C 180,E1 16774.158,E2 16774.158} C_VEL
LIN {X 0,Y 455.724,Z 786.317,A -85,B 0,C 180,E1 16773.352,E2 16773.352} C_VEL
LIN {X 0,Y 460.189,Z 762.664,A -85,B 0,C 180,E1 16772.57,E2 16772.57} C_VEL
LIN {X 0,Y 464.045,Z 736.24,A -85,B 0,C 180,E1 16771.916,E2 16771.916} C_VEL
LIN {X 0,Y 466.323,Z 713.85,A -85,B 0,C 180,E1 16771.488,E2 16771.488} C_VEL
LIN {X 0,Y 481.312,Z 484.14,A -85,B 0,C 180,E1 16767.848,E2 16767.848} C_VEL
LIN {X 0,Y 483.774,Z 445.949,A -85,B 0,C 180,E1 16767.226,E2 16767.226} C_VEL
LIN {X 0,Y 475.333,Z 431.084,A -85,B 0,C 180,E1 16764.813,E2 16764.813} C_VEL
LIN {X 0,Y 466.88,Z 417.219,A -85,B 0,C 180,E1 16762.111,E2 16762.111} C_VEL
LIN {X 0,Y 459.219,Z 406.521,A -85,B 0,C 180,E1 16759.36,E2 16759.36} C_VEL
LIN {X 0,Y 455.291,Z 401.193,A -85,B 0,C 180,E1 16757.774,E2 16757.774} C_VEL
LIN {X 0,Y 452.53,Z 397.43,A -85,B 0,C 180,E1 16756.561,E2 16756.561} C_VEL
LIN {X 0,Y 448.95,Z 392.666,A -85,B 0,C 180,E1 16754.84,E2 16754.84} C_VEL
LIN {X 0,Y 445.299,Z 387.72,A -85,B 0,C 180,E1 16752.844,E2 16752.844} C_VEL
LIN {X 0,Y 441.897,Z 383.476,A -85,B 0,C 180,E1 16750.693,E2 16750.693} C_VEL
LIN {X 0,Y 441.018,Z 382.205,A -85,B 0,C 180,E1 16750.054,E2 16750.054} C_VEL
LIN {X 0,Y 437.743,Z 378.395,A -85,B 0,C 180,E1 16747.349,E2 16747.349} C_VEL
LIN {X 0,Y 436.808,Z 376.507,A -85,B 0,C 180,E1 16746.308,E2 16746.308} C_VEL
LIN {X 0,Y 433.19,Z 372.596,A -85,B 0,C 180,E1 16739.074,E2 16739.074} C_VEL
LIN {X 0,Y 433.338,Z 372.983,A -85,B 0,C 180,E1 16736.561,E2 16736.561} C_VEL
LIN {X 0,Y 437.045,Z 376.827,A -85,B 0,C 180,E1 16730.253,E2 16730.253} C_VEL
LIN {X 0,Y 439.312,Z 380.623,A -85,B 0,C 180,E1 16728.046,E2 16728.046} C_VEL
LIN {X 0,Y 441.645,Z 383.006,A -85,B 0,C 180,E1 16726.315,E2 16726.315} C_VEL
LIN {X 0,Y 444.871,Z 387.321,A -85,B 0,C 180,E1 16724.219,E2 16724.219} C_VEL
LIN {X 0,Y 446.181,Z 388.952,A -85,B 0,C 180,E1 16723.465,E2 16723.465} C_VEL
LIN {X 0,Y 450.473,Z 394.686,A -85,B 0,C 180,E1 16721.225,E2 16721.225} C_VEL
LIN {X 0,Y 454.78,Z 400.401,A -85,B 0,C 180,E1 16719.269,E2 16719.269} C_VEL
LIN {X 0,Y 459.133,Z 406.344,A -85,B 0,C 180,E1 16717.496,E2 16717.496} C_VEL
LIN {X 0,Y 466.451,Z 416.681,A -85,B 0,C 180,E1 16714.851,E2 16714.851} C_VEL
LIN {X 0,Y 473.333,Z 426.804,A -85,B 0,C 180,E1 16712.648,E2 16712.648} C_VEL
LIN {X 0,Y 482.152,Z 440.63,A -85,B 0,C 180,E1 16710.113,E2 16710.113} C_VEL
LIN {X 0,Y 483.905,Z 443.89,A -85,B 0,C 180,E1 16709.629,E2 16709.629} C_VEL
LIN {X 0,Y 469.774,Z 659.87,A -85,B 0,C 180,E1 16706.217,E2 16706.217} C_VEL
LIN {X 0,Y 465.906,Z 716.6,A -85,B 0,C 180,E1 16705.295,E2 16705.295} C_VEL
LIN {X 0,Y 462.632,Z 743.651,A -85,B 0,C 180,E1 16704.709,E2 16704.709} C_VEL
LIN {X 0,Y 459.286,Z 764.344,A -85,B 0,C 180,E1 16704.126,E2 16704.126} C_VEL
LIN {X 0,Y 454.935,Z 786.734,A -85,B 0,C 180,E1 16703.342,E2 16703.342} C_VEL
LIN {X 0,Y 449.04,Z 812.046,A -85,B 0,C 180,E1 16702.231,E2 16702.231} C_VEL
LIN {X 0,Y 443.59,Z 832.293,A -85,B 0,C 180,E1 16701.149,E2 16701.149} C_VEL
LIN {X 0,Y 437.748,Z 851.863,A -85,B 0,C 180,E1 16699.924,E2 16699.924} C_VEL
LIN {X 0,Y 429.981,Z 875.312,A -85,B 0,C 180,E1 16698.184,E2 16698.184} C_VEL
LIN {X 0,Y 423.074,Z 894.243,A -85,B 0,C 180,E1 16696.515,E2 16696.515} C_VEL
LIN {X 0,Y 416.563,Z 911.065,A -85,B 0,C 180,E1 16694.808,E2 16694.808} C_VEL
LIN {X 0,Y 408.539,Z 930.773,A -85,B 0,C 180,E1 16692.493,E2 16692.493} C_VEL
LIN {X 0,Y 400.861,Z 948.449,A -85,B 0,C 180,E1 16690.024,E2 16690.024} C_VEL
LIN {X 0,Y 394.37,Z 963.106,A -85,B 0,C 180,E1 16687.664,E2 16687.664} C_VEL
LIN {X 0,Y 387.124,Z 979.376,A -85,B 0,C 180,E1 16684.627,E2 16684.627} C_VEL
LIN {X 0,Y 380.791,Z 993.44,A -85,B 0,C 180,E1 16681.502,E2 16681.502} C_VEL
LIN {X 0,Y 375.844,Z 1004.733,A -85,B 0,C 180,E1 16678.606,E2 16678.606} C_VEL
LIN {X 0,Y 370.717,Z 1017.144,A -85,B 0,C 180,E1 16674.882,E2 16674.882} C_VEL
LIN {X 0,Y 366.859,Z 1027.129,A -85,B 0,C 180,E1 16671.253,E2 16671.253} C_VEL
LIN {X 0,Y 364.214,Z 1034.919,A -85,B 0,C 180,E1 16667.907,E2 16667.907} C_VEL
LIN {X 0,Y 361.988,Z 1042.86,A -85,B 0,C 180,E1 16663.742,E2 16663.742} C_VEL
LIN {X 0,Y 360.802,Z 1048.274,A -85,B 0,C 180,E1 16660.055,E2 16660.055} C_VEL
LIN {X 0,Y 360.243,Z 1051.914,A -85,B 0,C 180,E1 16656.855,E2 16656.855} C_VEL
LIN {X 0,Y 359.999,Z 1054.559,A -85,B 0,C 180,E1 16653.663,E2 16653.663} C_VEL
LIN {X 0,Y 359.941,Z 1056.428,A -85,B 0,C 180,E1 16650,E2 16650} C_VEL
LIN {X 0,Y 359.907,Z 1056.934,A -85,B 0,C 180,E1 16646.177,E2 16646.177} C_VEL
LIN {X 0,Y 359.939,Z 1056.2,A -85,B 0,C 180,E1 16642.819,E2 16642.819} C_VEL
LIN {X 0,Y 360.045,Z 1054.504,A -85,B 0,C 180,E1 16639.6,E2 16639.6} C_VEL
LIN {X 0,Y 360.349,Z 1051.809,A -85,B 0,C 180,E1 16636.358,E2 16636.358} C_VEL
LIN {X 0,Y 361.081,Z 1047.884,A -85,B 0,C 180,E1 16632.931,E2 16632.931} C_VEL
LIN {X 0,Y 362.76,Z 1041.394,A -85,B 0,C 180,E1 16628.664,E2 16628.664} C_VEL
LIN {X 0,Y 365.048,Z 1034.33,A -85,B 0,C 180,E1 16625.044,E2 16625.044} C_VEL
LIN {X 0,Y 367.77,Z 1027.089,A -85,B 0,C 180,E1 16621.925,E2 16621.925} C_VEL
LIN {X 0,Y 367.96,Z 1024.454,A -85,B 0,C 180,E1 16620.79,E2 16620.79} C_VEL
LIN {X 0,Y 365.426,Z 1017.237,A -85,B 0,C 180,E1 16617.688,E2 16617.688} C_VEL
LIN {X 0,Y 365.998,Z 1014.49,A -85,B 0,C 180,E1 16616.74,E2 16616.74} C_VEL
LIN {X 0,Y 371.223,Z 1003.539,A -85,B 0,C 180,E1 16613.469,E2 16613.469} C_VEL
LIN {X 0,Y 377.355,Z 991.242,A -85,B 0,C 180,E1 16610.314,E2 16610.314} C_VEL
LIN {X 0,Y 385.194,Z 975.637,A -85,B 0,C 180,E1 16606.945,E2 16606.945} C_VEL
LIN {X 0,Y 392.022,Z 961.935,A -85,B 0,C 180,E1 16604.425,E2 16604.425} C_VEL
LIN {X 0,Y 399.514,Z 946.649,A -85,B 0,C 180,E1 16601.985,E2 16601.985} C_VEL
LIN {X 0,Y 408.818,Z 926.849,A -85,B 0,C 180,E1 16599.306,E2 16599.306} C_VEL
LIN {X 0,Y 416.651,Z 909.241,A -85,B 0,C 180,E1 16597.294,E2 16597.294} C_VEL
LIN {X 0,Y 424.611,Z 890.343,A -85,B 0,C 180,E1 16595.435,E2 16595.435} C_VEL
LIN {X 0,Y 433.249,Z 867.855,A -85,B 0,C 180,E1 16593.577,E2 16593.577} C_VEL
LIN {X 0,Y 439.873,Z 849.012,A -85,B 0,C 180,E1 16592.264,E2 16592.264} C_VEL
LIN {X 0,Y 446.075,Z 829.617,A -85,B 0,C 180,E1 16591.101,E2 16591.101} C_VEL
LIN {X 0,Y 453.091,Z 804.706,A -85,B 0,C 180,E1 16589.856,E2 16589.856} C_VEL
LIN {X 0,Y 458.301,Z 782.865,A -85,B 0,C 180,E1 16588.97,E2 16588.97} C_VEL
LIN {X 0,Y 462.774,Z 760.831,A -85,B 0,C 180,E1 16588.239,E2 16588.239} C_VEL
LIN {X 0,Y 467.291,Z 732.525,A -85,B 0,C 180,E1 16587.527,E2 16587.527} C_VEL
LIN {X 0,Y 469.785,Z 710.082,A -85,B 0,C 180,E1 16587.103,E2 16587.103} C_VEL
LIN {X 0,Y 486.305,Z 480.738,A -85,B 0,C 180,E1 16583.492,E2 16583.492} C_VEL
LIN {X 0,Y 488.269,Z 453.17,A -85,B 0,C 180,E1 16583.043,E2 16583.043} C_VEL
LIN {X 0,Y 481.389,Z 442.246,A -85,B 0,C 180,E1 16580.773,E2 16580.773} C_VEL
LIN {X 0,Y 474.861,Z 432.437,A -85,B 0,C 180,E1 16578.349,E2 16578.349} C_VEL
LIN {X 0,Y 468.857,Z 423.77,A -85,B 0,C 180,E1 16575.778,E2 16575.778} C_VEL
LIN {X 0,Y 465.568,Z 419.156,A -85,B 0,C 180,E1 16574.172,E2 16574.172} C_VEL
LIN {X 0,Y 462.387,Z 414.718,A -85,B 0,C 180,E1 16572.425,E2 16572.425} C_VEL
LIN {X 0,Y 458.877,Z 409.79,A -85,B 0,C 180,E1 16570.166,E2 16570.166} C_VEL
LIN {X 0,Y 455.758,Z 405.66,A -85,B 0,C 180,E1 16567.691,E2 16567.691} C_VEL
LIN {X 0,Y 454.99,Z 404.415,A -85,B 0,C 180,E1 16566.942,E2 16566.942} C_VEL
LIN {X 0,Y 452.151,Z 401.023,A -85,B 0,C 180,E1 16563.423,E2 16563.423} C_VEL
LIN {X 0,Y 451.464,Z 399.104,A -85,B 0,C 180,E1 16561.777,E2 16561.777} C_VEL
LIN {X 0,Y 450.874,Z 398.699,A -85,B 0,C 180,E1 16557.458,E2 16557.458} C_VEL
LIN {X 0,Y 451.619,Z 399.375,A -85,B 0,C 180,E1 16554.919,E2 16554.919} C_VEL
LIN {X 0,Y 453.993,Z 403.71,A -85,B 0,C 180,E1 16551.131,E2 16551.131} C_VEL
LIN {X 0,Y 455.533,Z 405.118,A -85,B 0,C 180,E1 16549.631,E2 16549.631} C_VEL
LIN {X 0,Y 458.555,Z 409.478,A -85,B 0,C 180,E1 16547.149,E2 16547.149} C_VEL
LIN {X 0,Y 459.703,Z 411.047,A -85,B 0,C 180,E1 16546.35,E2 16546.35} C_VEL
LIN {X 0,Y 463.719,Z 416.497,A -85,B 0,C 180,E1 16543.914,E2 16543.914} C_VEL
LIN {X 0,Y 467.42,Z 421.775,A -85,B 0,C 180,E1 16541.994,E2 16541.994} C_VEL
LIN {X 0,Y 472.117,Z 428.495,A -85,B 0,C 180,E1 16539.87,E2 16539.87} C_VEL
LIN {X 0,Y 476.924,Z 435.91,A -85,B 0,C 180,E1 16537.928,E2 16537.928} C_VEL
LIN {X 0,Y 484.852,Z 449.273,A -85,B 0,C 180,E1 16535.088,E2 16535.088} C_VEL
LIN {X 0,Y 488.23,Z 455.669,A -85,B 0,C 180,E1 16533.976,E2 16533.976} C_VEL
LIN {X 0,Y 471.772,Z 685.149,A -85,B 0,C 180,E1 16530.374,E2 16530.374} C_VEL
LIN {X 0,Y 468.599,Z 725.185,A -85,B 0,C 180,E1 16529.713,E2 16529.713} C_VEL
LIN {X 0,Y 465.136,Z 750.164,A -85,B 0,C 180,E1 16529.173,E2 16529.173} C_VEL
LIN {X 0,Y 461.26,Z 771.778,A -85,B 0,C 180,E1 16528.584,E2 16528.584} C_VEL
LIN {X 0,Y 455.589,Z 797.844,A -85,B 0,C 180,E1 16527.668,E2 16527.668} C_VEL
LIN {X 0,Y 449.83,Z 819.808,A -85,B 0,C 180,E1 16526.697,E2 16526.697} C_VEL
LIN {X 0,Y 443.926,Z 839.829,A -85,B 0,C 180,E1 16525.638,E2 16525.638} C_VEL
LIN {X 0,Y 436.389,Z 862.74,A -85,B 0,C 180,E1 16524.204,E2 16524.204} C_VEL
LIN {X 0,Y 428.533,Z 883.867,A -85,B 0,C 180,E1 16522.606,E2 16522.606} C_VEL
LIN {X 0,Y 421.47,Z 901.554,A -85,B 0,C 180,E1 16521.047,E2 16521.047} C_VEL
LIN {X 0,Y 412.976,Z 921.589,A -85,B 0,C 180,E1 16518.994,E2 16518.994} C_VEL
LIN {X 0,Y 404.23,Z 940.668,A -85,B 0,C 180,E1 16516.654,E2 16516.654} C_VEL
LIN {X 0,Y 397.301,Z 955.271,A -85,B 0,C 180,E1 16514.583,E2 16514.583} C_VEL
LIN {X 0,Y 389.725,Z 970.876,A -85,B 0,C 180,E1 16512.038,E2 16512.038} C_VEL
LIN {X 0,Y 381.387,Z 987.659,A -85,B 0,C 180,E1 16508.799,E2 16508.799} C_VEL
LIN {X 0,Y 375.09,Z 1000.386,A -85,B 0,C 180,E1 16505.906,E2 16505.906} C_VEL
LIN {X 0,Y 368.854,Z 1013.422,A -85,B 0,C 180,E1 16502.462,E2 16502.462} C_VEL
LIN {X 0,Y 363.228,Z 1025.599,A -85,B 0,C 180,E1 16498.581,E2 16498.581} C_VEL
LIN {X 0,Y 359.452,Z 1034.583,A -85,B 0,C 180,E1 16495.189,E2 16495.189} C_VEL
LIN {X 0,Y 356.203,Z 1043.423,A -85,B 0,C 180,E1 16491.23,E2 16491.23} C_VEL
LIN {X 0,Y 353.946,Z 1050.691,A -85,B 0,C 180,E1 16487.085,E2 16487.085} C_VEL
LIN {X 0,Y 352.844,Z 1055.362,A -85,B 0,C 180,E1 16483.771,E2 16483.771} C_VEL
LIN {X 0,Y 352.23,Z 1058.997,A -85,B 0,C 180,E1 16480.468,E2 16480.468} C_VEL
LIN {X 0,Y 351.967,Z 1061.964,A -85,B 0,C 180,E1 16476.689,E2 16476.689} C_VEL
LIN {X 0,Y 351.912,Z 1063.604,A -85,B 0,C 180,E1 16472.606,E2 16472.606} C_VEL
LIN {X 0,Y 351.913,Z 1063.799,A -85,B 0,C 180,E1 16469.349,E2 16469.349} C_VEL
LIN {X 0,Y 351.913,Z 1063.001,A -85,B 0,C 180,E1 16466.09,E2 16466.09} C_VEL
LIN {X 0,Y 351.985,Z 1061.204,A -85,B 0,C 180,E1 16462.82,E2 16462.82} C_VEL
LIN {X 0,Y 352.219,Z 1058.394,A -85,B 0,C 180,E1 16459.532,E2 16459.532} C_VEL
LIN {X 0,Y 352.965,Z 1053.83,A -85,B 0,C 180,E1 16455.658,E2 16455.658} C_VEL
LIN {X 0,Y 354.56,Z 1047.021,A -85,B 0,C 180,E1 16451.418,E2 16451.418} C_VEL
LIN {X 0,Y 356.66,Z 1040.08,A -85,B 0,C 180,E1 16447.935,E2 16447.935} C_VEL
LIN {X 0,Y 360.093,Z 1030.63,A -85,B 0,C 180,E1 16443.978,E2 16443.978} C_VEL
LIN {X 0,Y 364.475,Z 1019.633,A -85,B 0,C 180,E1 16440.228,E2 16440.228} C_VEL
LIN {X 0,Y 369.077,Z 1008.997,A -85,B 0,C 180,E1 16437.124,E2 16437.124} C_VEL
LIN {X 0,Y 375.233,Z 995.504,A -85,B 0,C 180,E1 16433.732,E2 16433.732} C_VEL
LIN {X 0,Y 382.281,Z 980.092,A -85,B 0,C 180,E1 16430.498,E2 16430.498} C_VEL
LIN {X 0,Y 388.593,Z 966.374,A -85,B 0,C 180,E1 16428.01,E2 16428.01} C_VEL
LIN {X 0,Y 396.492,Z 949.04,A -85,B 0,C 180,E1 16425.284,E2 16425.284} C_VEL
LIN {X 0,Y 404.669,Z 930.103,A -85,B 0,C 180,E1 16422.79,E2 16422.79} C_VEL
LIN {X 0,Y 411.776,Z 913.027,A -85,B 0,C 180,E1 16420.853,E2 16420.853} C_VEL
LIN {X 0,Y 420.118,Z 891.808,A -85,B 0,C 180,E1 16418.79,E2 16418.79} C_VEL
LIN {X 0,Y 427.518,Z 871.112,A -85,B 0,C 180,E1 16417.105,E2 16417.105} C_VEL
LIN {X 0,Y 433.832,Z 852.076,A -85,B 0,C 180,E1 16415.779,E2 16415.779} C_VEL
LIN {X 0,Y 440.674,Z 829.393,A -85,B 0,C 180,E1 16414.434,E2 16414.434} C_VEL
LIN {X 0,Y 446.784,Z 805.708,A -85,B 0,C 180,E1 16413.293,E2 16413.293} C_VEL
LIN {X 0,Y 451.169,Z 786.319,A -85,B 0,C 180,E1 16412.513,E2 16412.513} C_VEL
LIN {X 0,Y 455.669,Z 763.02,A -85,B 0,C 180,E1 16411.744,E2 16411.744} C_VEL
LIN {X 0,Y 459.651,Z 736.477,A -85,B 0,C 180,E1 16411.086,E2 16411.086} C_VEL
LIN {X 0,Y 461.993,Z 714.076,A -85,B 0,C 180,E1 16410.657,E2 16410.657} C_VEL
LIN {X 0,Y 477.394,Z 484.773,A -85,B 0,C 180,E1 16407.017,E2 16407.017} C_VEL
LIN {X 0,Y 479.692,Z 450.335,A -85,B 0,C 180,E1 16406.459,E2 16406.459} C_VEL
LIN {X 0,Y 472.347,Z 437.197,A -85,B 0,C 180,E1 16404.28,E2 16404.28} C_VEL
LIN {X 0,Y 464.506,Z 424.119,A -85,B 0,C 180,E1 16401.698,E2 16401.698} C_VEL
LIN {X 0,Y 457.079,Z 413.559,A -85,B 0,C 180,E1 16398.957,E2 16398.957} C_VEL
LIN {X 0,Y 451.415,Z 405.587,A -85,B 0,C 180,E1 16396.537,E2 16396.537} C_VEL
LIN {X 0,Y 447.355,Z 400.214,A -85,B 0,C 180,E1 16394.563,E2 16394.563} C_VEL
LIN {X 0,Y 443.664,Z 395.215,A -85,B 0,C 180,E1 16392.495,E2 16392.495} C_VEL
LIN {X 0,Y 440.379,Z 390.854,A -85,B 0,C 180,E1 16390.333,E2 16390.333} C_VEL
LIN {X 0,Y 439.328,Z 389.658,A -85,B 0,C 180,E1 16389.564,E2 16389.564} C_VEL
LIN {X 0,Y 436.322,Z 385.715,A -85,B 0,C 180,E1 16386.91,E2 16386.91} C_VEL
LIN {X 0,Y 435.582,Z 384.331,A -85,B 0,C 180,E1 16386.061,E2 16386.061} C_VEL
LIN {X 0,Y 432.214,Z 380.538,A -85,B 0,C 180,E1 16379.072,E2 16379.072} C_VEL
LIN {X 0,Y 432.361,Z 380.948,A -85,B 0,C 180,E1 16376.553,E2 16376.553} C_VEL
LIN {X 0,Y 435.886,Z 384.666,A -85,B 0,C 180,E1 16370.427,E2 16370.427} C_VEL
LIN {X 0,Y 438.185,Z 388.514,A -85,B 0,C 180,E1 16368.149,E2 16368.149} C_VEL
LIN {X 0,Y 440.31,Z 390.719,A -85,B 0,C 180,E1 16366.54,E2 16366.54} C_VEL
LIN {X 0,Y 443.584,Z 395.126,A -85,B 0,C 180,E1 16364.373,E2 16364.373} C_VEL
LIN {X 0,Y 445.189,Z 397.379,A -85,B 0,C 180,E1 16363.427,E2 16363.427} C_VEL
LIN {X 0,Y 448.862,Z 402.249,A -85,B 0,C 180,E1 16361.492,E2 16361.492} C_VEL
LIN {X 0,Y 453.098,Z 407.973,A -85,B 0,C 180,E1 16359.526,E2 16359.526} C_VEL
LIN {X 0,Y 458.703,Z 415.658,A -85,B 0,C 180,E1 16357.237,E2 16357.237} C_VEL
LIN {X 0,Y 467.907,Z 429.112,A -85,B 0,C 180,E1 16353.985,E2 16353.985} C_VEL
LIN {X 0,Y 476.685,Z 442.918,A -85,B 0,C 180,E1 16351.292,E2 16351.292} C_VEL
LIN {X 0,Y 479.812,Z 448.186,A -85,B 0,C 180,E1 16350.402,E2 16350.402} C_VEL
LIN {X 0,Y 465.017,Z 668.302,A -85,B 0,C 180,E1 16346.92,E2 16346.92} C_VEL
LIN {X 0,Y 461.462,Z 718.163,A -85,B 0,C 180,E1 16346.103,E2 16346.103} C_VEL
LIN {X 0,Y 458.13,Z 744.447,A -85,B 0,C 180,E1 16345.526,E2 16345.526} C_VEL
LIN {X 0,Y 454.734,Z 764.892,A -85,B 0,C 180,E1 16344.949,E2 16344.949} C_VEL
LIN {X 0,Y 450.225,Z 787.51,A -85,B 0,C 180,E1 16344.156,E2 16344.156} C_VEL
LIN {X 0,Y 444.189,Z 812.659,A -85,B 0,C 180,E1 16343.046,E2 16343.046} C_VEL
LIN {X 0,Y 438.609,Z 832.848,A -85,B 0,C 180,E1 16341.964,E2 16341.964} C_VEL
LIN {X 0,Y 432.622,Z 852.369,A -85,B 0,C 180,E1 16340.738,E2 16340.738} C_VEL
LIN {X 0,Y 424.376,Z 876.469,A -85,B 0,C 180,E1 16338.935,E2 16338.935} C_VEL
LIN {X 0,Y 417.294,Z 895.305,A -85,B 0,C 180,E1 16337.257,E2 16337.257} C_VEL
LIN {X 0,Y 410.317,Z 912.759,A -85,B 0,C 180,E1 16335.462,E2 16335.462} C_VEL
LIN {X 0,Y 401.206,Z 934.1,A -85,B 0,C 180,E1 16332.872,E2 16332.872} C_VEL
LIN {X 0,Y 394.305,Z 949.513,A -85,B 0,C 180,E1 16330.67,E2 16330.67} C_VEL
LIN {X 0,Y 387.176,Z 965.063,A -85,B 0,C 180,E1 16328.113,E2 16328.113} C_VEL
LIN {X 0,Y 379.409,Z 981.703,A -85,B 0,C 180,E1 16324.881,E2 16324.881} C_VEL
LIN {X 0,Y 373.537,Z 994.305,A -85,B 0,C 180,E1 16322.006,E2 16322.006} C_VEL
LIN {X 0,Y 367.938,Z 1006.637,A -85,B 0,C 180,E1 16318.751,E2 16318.751} C_VEL
LIN {X 0,Y 362.639,Z 1018.866,A -85,B 0,C 180,E1 16314.886,E2 16314.886} C_VEL
LIN {X 0,Y 359.105,Z 1027.71,A -85,B 0,C 180,E1 16311.564,E2 16311.564} C_VEL
LIN {X 0,Y 356.145,Z 1036.133,A -85,B 0,C 180,E1 16307.819,E2 16307.819} C_VEL
LIN {X 0,Y 353.909,Z 1043.756,A -85,B 0,C 180,E1 16303.562,E2 16303.562} C_VEL
LIN {X 0,Y 352.82,Z 1048.609,A -85,B 0,C 180,E1 16300.12,E2 16300.12} C_VEL
LIN {X 0,Y 352.225,Z 1052.349,A -85,B 0,C 180,E1 16296.684,E2 16296.684} C_VEL
LIN {X 0,Y 351.958,Z 1055.341,A -85,B 0,C 180,E1 16292.768,E2 16292.768} C_VEL
LIN {X 0,Y 351.913,Z 1056.755,A -85,B 0,C 180,E1 16289.023,E2 16289.023} C_VEL
LIN {X 0,Y 351.908,Z 1056.939,A -85,B 0,C 180,E1 16285.6,E2 16285.6} C_VEL
LIN {X 0,Y 351.933,Z 1056.193,A -85,B 0,C 180,E1 16282.49,E2 16282.49} C_VEL
LIN {X 0,Y 352.072,Z 1054.441,A -85,B 0,C 180,E1 16279.197,E2 16279.197} C_VEL
LIN {X 0,Y 352.432,Z 1051.688,A -85,B 0,C 180,E1 16275.878,E2 16275.878} C_VEL
LIN {X 0,Y 353.411,Z 1047.152,A -85,B 0,C 180,E1 16271.922,E2 16271.922} C_VEL
LIN {X 0,Y 355.297,Z 1040.486,A -85,B 0,C 180,E1 16267.671,E2 16267.671} C_VEL
LIN {X 0,Y 357.731,Z 1033.625,A -85,B 0,C 180,E1 16264.149,E2 16264.149} C_VEL
LIN {X 0,Y 361.623,Z 1024.259,A -85,B 0,C 180,E1 16260.152,E2 16260.152} C_VEL
LIN {X 0,Y 365.998,Z 1014.49,A -85,B 0,C 180,E1 16256.74,E2 16256.74} C_VEL
LIN {X 0,Y 366.631,Z 1011.298,A -85,B 0,C 180,E1 16255.642,E2 16255.642} C_VEL
LIN {X 0,Y 365.39,Z 1002.924,A -85,B 0,C 180,E1 16252.588,E2 16252.588} C_VEL
LIN {X 0,Y 366.39,Z 999.87,A -85,B 0,C 180,E1 16251.671,E2 16251.671} C_VEL
LIN {X 0,Y 373.73,Z 985.704,A -85,B 0,C 180,E1 16248.227,E2 16248.227} C_VEL
LIN {X 0,Y 380.667,Z 972.419,A -85,B 0,C 180,E1 16245.467,E2 16245.467} C_VEL
LIN {X 0,Y 389.389,Z 955.639,A -85,B 0,C 180,E1 16242.481,E2 16242.481} C_VEL
LIN {X 0,Y 398.064,Z 938.095,A -85,B 0,C 180,E1 16239.881,E2 16239.881} C_VEL
LIN {X 0,Y 405.551,Z 922.4,A -85,B 0,C 180,E1 16237.873,E2 16237.873} C_VEL
LIN {X 0,Y 414.73,Z 902.229,A -85,B 0,C 180,E1 16235.661,E2 16235.661} C_VEL
LIN {X 0,Y 423.052,Z 882.142,A -85,B 0,C 180,E1 16233.822,E2 16233.822} C_VEL
LIN {X 0,Y 430.242,Z 863.441,A -85,B 0,C 180,E1 16232.352,E2 16232.352} C_VEL
LIN {X 0,Y 438.368,Z 840.384,A -85,B 0,C 180,E1 16230.821,E2 16230.821} C_VEL
LIN {X 0,Y 445.389,Z 817.345,A -85,B 0,C 180,E1 16229.567,E2 16229.567} C_VEL
LIN {X 0,Y 451.061,Z 796.378,A -85,B 0,C 180,E1 16228.618,E2 16228.618} C_VEL
LIN {X 0,Y 456.903,Z 770.921,A -85,B 0,C 180,E1 16227.681,E2 16227.681} C_VEL
LIN {X 0,Y 461.023,Z 748.512,A -85,B 0,C 180,E1 16227.037,E2 16227.037} C_VEL
LIN {X 0,Y 464.172,Z 726.937,A -85,B 0,C 180,E1 16226.547,E2 16226.547} C_VEL
LIN {X 0,Y 466.9,Z 699.501,A -85,B 0,C 180,E1 16226.059,E2 16226.059} C_VEL
LIN {X 0,Y 483.685,Z 471.02,A -85,B 0,C 180,E1 16222.475,E2 16222.475} C_VEL
LIN {X 0,Y 484.598,Z 457.917,A -85,B 0,C 180,E1 16222.249,E2 16222.249} C_VEL
LIN {X 0,Y 476.459,Z 444.985,A -85,B 0,C 180,E1 16219.396,E2 16219.396} C_VEL
LIN {X 0,Y 470.21,Z 435.704,A -85,B 0,C 180,E1 16216.874,E2 16216.874} C_VEL
LIN {X 0,Y 464.945,Z 427.823,A -85,B 0,C 180,E1 16214.382,E2 16214.382} C_VEL
LIN {X 0,Y 460.777,Z 422.172,A -85,B 0,C 180,E1 16212.088,E2 16212.088} C_VEL
LIN {X 0,Y 457.543,Z 417.503,A -85,B 0,C 180,E1 16209.942,E2 16209.942} C_VEL
LIN {X 0,Y 454.446,Z 413.211,A -85,B 0,C 180,E1 16207.395,E2 16207.395} C_VEL
LIN {X 0,Y 453.752,Z 412.198,A -85,B 0,C 180,E1 16206.707,E2 16206.707} C_VEL
LIN {X 0,Y 451.036,Z 408.752,A -85,B 0,C 180,E1 16203.177,E2 16203.177} C_VEL
LIN {X 0,Y 450.439,Z 407.004,A -85,B 0,C 180,E1 16201.654,E2 16201.654} C_VEL
LIN {X 0,Y 449.918,Z 406.658,A -85,B 0,C 180,E1 16197.325,E2 16197.325} C_VEL
LIN {X 0,Y 450.59,Z 407.269,A -85,B 0,C 180,E1 16195.035,E2 16195.035} C_VEL
LIN {X 0,Y 452.907,Z 411.592,A -85,B 0,C 180,E1 16191.238,E2 16191.238} C_VEL
LIN {X 0,Y 454.355,Z 412.949,A -85,B 0,C 180,E1 16189.796,E2 16189.796} C_VEL
LIN {X 0,Y 457.412,Z 417.37,A -85,B 0,C 180,E1 16187.245,E2 16187.245} C_VEL
LIN {X 0,Y 462.198,Z 424.049,A -85,B 0,C 180,E1 16184.182,E2 16184.182} C_VEL
LIN {X 0,Y 465.945,Z 429.523,A -85,B 0,C 180,E1 16182.194,E2 16182.194} C_VEL
LIN {X 0,Y 471.484,Z 437.498,A -85,B 0,C 180,E1 16179.679,E2 16179.679} C_VEL
LIN {X 0,Y 477.575,Z 447.624,A -85,B 0,C 180,E1 16177.244,E2 16177.244} C_VEL
LIN {X 0,Y 484.23,Z 459.373,A -85,B 0,C 180,E1 16174.891,E2 16174.891} C_VEL
LIN {X 0,Y 484.57,Z 460.374,A -85,B 0,C 180,E1 16174.764,E2 16174.764} C_VEL
LIN {X 0,Y 467.662,Z 690.17,A -85,B 0,C 180,E1 16171.159,E2 16171.159} C_VEL
LIN {X 0,Y 464.597,Z 726.418,A -85,B 0,C 180,E1 16170.554,E2 16170.554} C_VEL
LIN {X 0,Y 461.189,Z 750.362,A -85,B 0,C 180,E1 16170.036,E2 16170.036} C_VEL
LIN {X 0,Y 457.191,Z 772.143,A -85,B 0,C 180,E1 16169.445,E2 16169.445} C_VEL
LIN {X 0,Y 451.353,Z 798.255,A -85,B 0,C 180,E1 16168.528,E2 16168.528} C_VEL
LIN {X 0,Y 445.432,Z 820.288,A -85,B 0,C 180,E1 16167.554,E2 16167.554} C_VEL
LIN {X 0,Y 439.426,Z 840.135,A -85,B 0,C 180,E1 16166.506,E2 16166.506} C_VEL
LIN {X 0,Y 431.702,Z 862.972,A -85,B 0,C 180,E1 16165.076,E2 16165.076} C_VEL
LIN {X 0,Y 423.641,Z 884.067,A -85,B 0,C 180,E1 16163.481,E2 16163.481} C_VEL
LIN {X 0,Y 416.492,Z 901.46,A -85,B 0,C 180,E1 16161.947,E2 16161.947} C_VEL
LIN {X 0,Y 407.803,Z 921.359,A -85,B 0,C 180,E1 16159.906,E2 16159.906} C_VEL
LIN {X 0,Y 398.962,Z 940.081,A -85,B 0,C 180,E1 16157.61,E2 16157.61} C_VEL
LIN {X 0,Y 391.494,Z 955.287,A -85,B 0,C 180,E1 16155.445,E2 16155.445} C_VEL
LIN {X 0,Y 383.612,Z 970.955,A -85,B 0,C 180,E1 16152.867,E2 16152.867} C_VEL
LIN {X 0,Y 374.907,Z 987.793,A -85,B 0,C 180,E1 16149.576,E2 16149.576} C_VEL
LIN {X 0,Y 368.381,Z 1000.424,A -85,B 0,C 180,E1 16146.665,E2 16146.665} C_VEL
LIN {X 0,Y 361.802,Z 1013.57,A -85,B 0,C 180,E1 16143.135,E2 16143.135} C_VEL
LIN {X 0,Y 355.991,Z 1025.504,A -85,B 0,C 180,E1 16139.256,E2 16139.256} C_VEL
LIN {X 0,Y 351.969,Z 1034.576,A -85,B 0,C 180,E1 16135.763,E2 16135.763} C_VEL
LIN {X 0,Y 348.399,Z 1043.715,A -85,B 0,C 180,E1 16131.552,E2 16131.552} C_VEL
LIN {X 0,Y 346.103,Z 1050.657,A -85,B 0,C 180,E1 16127.485,E2 16127.485} C_VEL
LIN {X 0,Y 344.881,Z 1055.526,A -85,B 0,C 180,E1 16123.924,E2 16123.924} C_VEL
LIN {X 0,Y 344.219,Z 1059.268,A -85,B 0,C 180,E1 16120.375,E2 16120.375} C_VEL
LIN {X 0,Y 343.943,Z 1062.283,A -85,B 0,C 180,E1 16116.175,E2 16116.175} C_VEL
LIN {X 0,Y 343.911,Z 1063.553,A -85,B 0,C 180,E1 16112.5,E2 16112.5} C_VEL
LIN {X 0,Y 343.913,Z 1063.695,A -85,B 0,C 180,E1 16109.167,E2 16109.167} C_VEL
LIN {X 0,Y 343.912,Z 1062.911,A -85,B 0,C 180,E1 16105.999,E2 16105.999} C_VEL
LIN {X 0,Y 343.994,Z 1061.106,A -85,B 0,C 180,E1 16102.652,E2 16102.652} C_VEL
LIN {X 0,Y 344.249,Z 1058.287,A -85,B 0,C 180,E1 16099.287,E2 16099.287} C_VEL
LIN {X 0,Y 345.086,Z 1053.598,A -85,B 0,C 180,E1 16095.228,E2 16095.228} C_VEL
LIN {X 0,Y 346.762,Z 1046.886,A -85,B 0,C 180,E1 16090.984,E2 16090.984} C_VEL
LIN {X 0,Y 348.873,Z 1040.294,A -85,B 0,C 180,E1 16087.593,E2 16087.593} C_VEL
LIN {X 0,Y 352.114,Z 1031.706,A -85,B 0,C 180,E1 16083.887,E2 16083.887} C_VEL
LIN {X 0,Y 357.034,Z 1019.979,A -85,B 0,C 180,E1 16079.729,E2 16079.729} C_VEL
LIN {X 0,Y 361.791,Z 1009.433,A -85,B 0,C 180,E1 16076.579,E2 16076.579} C_VEL
LIN {X 0,Y 367.878,Z 996.59,A -85,B 0,C 180,E1 16073.277,E2 16073.277} C_VEL
LIN {X 0,Y 375.503,Z 980.639,A -85,B 0,C 180,E1 16069.838,E2 16069.838} C_VEL
LIN {X 0,Y 382.019,Z 966.987,A -85,B 0,C 180,E1 16067.32,E2 16067.32} C_VEL
LIN {X 0,Y 389.712,Z 950.659,A -85,B 0,C 180,E1 16064.708,E2 16064.708} C_VEL
LIN {X 0,Y 398.584,Z 930.935,A -85,B 0,C 180,E1 16062.052,E2 16062.052} C_VEL
LIN {X 0,Y 405.788,Z 914.173,A -85,B 0,C 180,E1 16060.126,E2 16060.126} C_VEL
LIN {X 0,Y 413.897,Z 894.285,A -85,B 0,C 180,E1 16058.156,E2 16058.156} C_VEL
LIN {X 0,Y 422.173,Z 871.95,A -85,B 0,C 180,E1 16056.307,E2 16056.307} C_VEL
LIN {X 0,Y 428.801,Z 852.514,A -85,B 0,C 180,E1 16054.946,E2 16054.946} C_VEL
LIN {X 0,Y 435.791,Z 829.969,A -85,B 0,C 180,E1 16053.605,E2 16053.605} C_VEL
LIN {X 0,Y 442.045,Z 806.432,A -85,B 0,C 180,E1 16052.466,E2 16052.466} C_VEL
LIN {X 0,Y 446.69,Z 786.415,A -85,B 0,C 180,E1 16051.662,E2 16051.662} C_VEL
LIN {X 0,Y 451.256,Z 763.321,A -85,B 0,C 180,E1 16050.901,E2 16050.901} C_VEL
LIN {X 0,Y 455.377,Z 736.545,A -85,B 0,C 180,E1 16050.237,E2 16050.237} C_VEL
LIN {X 0,Y 457.779,Z 714.081,A -85,B 0,C 180,E1 16049.807,E2 16049.807} C_VEL
LIN {X 0,Y 473.547,Z 485.815,A -85,B 0,C 180,E1 16046.18,E2 16046.18} C_VEL
LIN {X 0,Y 475.646,Z 454.547,A -85,B 0,C 180,E1 16045.661,E2 16045.661} C_VEL
LIN {X 0,Y 468.345,Z 441.431,A -85,B 0,C 180,E1 16043.397,E2 16043.397} C_VEL
LIN {X 0,Y 461.906,Z 430.665,A -85,B 0,C 180,E1 16041.193,E2 16041.193} C_VEL
LIN {X 0,Y 454.962,Z 420.594,A -85,B 0,C 180,E1 16038.55,E2 16038.55} C_VEL
LIN {X 0,Y 449.357,Z 412.658,A -85,B 0,C 180,E1 16036.083,E2 16036.083} C_VEL
LIN {X 0,Y 445.65,Z 407.624,A -85,B 0,C 180,E1 16034.222,E2 16034.222} C_VEL
LIN {X 0,Y 442.154,Z 402.802,A -85,B 0,C 180,E1 16032.207,E2 16032.207} C_VEL
LIN {X 0,Y 438.878,Z 398.23,A -85,B 0,C 180,E1 16029.971,E2 16029.971} C_VEL
LIN {X 0,Y 435.267,Z 393.761,A -85,B 0,C 180,E1 16026.861,E2 16026.861} C_VEL
LIN {X 0,Y 434.486,Z 392.222,A -85,B 0,C 180,E1 16025.944,E2 16025.944} C_VEL
LIN {X 0,Y 431.238,Z 388.481,A -85,B 0,C 180,E1 16019.07,E2 16019.07} C_VEL
LIN {X 0,Y 431.362,Z 388.838,A -85,B 0,C 180,E1 16016.678,E2 16016.678} C_VEL
LIN {X 0,Y 434.782,Z 392.637,A -85,B 0,C 180,E1 16010.536,E2 16010.536} C_VEL
LIN {X 0,Y 437.216,Z 396.574,A -85,B 0,C 180,E1 16008.122,E2 16008.122} C_VEL
LIN {X 0,Y 439.065,Z 398.586,A -85,B 0,C 180,E1 16006.702,E2 16006.702} C_VEL
LIN {X 0,Y 442.299,Z 402.932,A -85,B 0,C 180,E1 16004.528,E2 16004.528} C_VEL
LIN {X 0,Y 447.261,Z 409.81,A -85,B 0,C 180,E1 16001.761,E2 16001.761} C_VEL
LIN {X 0,Y 451.562,Z 415.739,A -85,B 0,C 180,E1 15999.724,E2 15999.724} C_VEL
LIN {X 0,Y 456.791,Z 423.06,A -85,B 0,C 180,E1 15997.544,E2 15997.544} C_VEL
LIN {X 0,Y 465.596,Z 436.147,A -85,B 0,C 180,E1 15994.359,E2 15994.359} C_VEL
LIN {X 0,Y 474.231,Z 449.976,A -85,B 0,C 180,E1 15991.645,E2 15991.645} C_VEL
LIN {X 0,Y 475.786,Z 452.792,A -85,B 0,C 180,E1 15991.182,E2 15991.182} C_VEL
LIN {X 0,Y 460.467,Z 674.695,A -85,B 0,C 180,E1 15987.67,E2 15987.67} C_VEL
LIN {X 0,Y 457.091,Z 719.886,A -85,B 0,C 180,E1 15986.924,E2 15986.924} C_VEL
LIN {X 0,Y 453.682,Z 745.493,A -85,B 0,C 180,E1 15986.353,E2 15986.353} C_VEL
LIN {X 0,Y 450.198,Z 765.872,A -85,B 0,C 180,E1 15985.775,E2 15985.775} C_VEL
LIN {X 0,Y 445.13,Z 790.577,A -85,B 0,C 180,E1 15984.897,E2 15984.897} C_VEL
LIN {X 0,Y 439.125,Z 814.387,A -85,B 0,C 180,E1 15983.823,E2 15983.823} C_VEL
LIN {X 0,Y 433.422,Z 834.396,A -85,B 0,C 180,E1 15982.74,E2 15982.74} C_VEL
LIN {X 0,Y 426.079,Z 857.498,A -85,B 0,C 180,E1 15981.26,E2 15981.26} C_VEL
LIN {X 0,Y 418.29,Z 879.075,A -85,B 0,C 180,E1 15979.583,E2 15979.583} C_VEL
LIN {X 0,Y 411.323,Z 897.022,A -85,B 0,C 180,E1 15977.957,E2 15977.957} C_VEL
LIN {X 0,Y 402.934,Z 917.284,A -85,B 0,C 180,E1 15975.82,E2 15975.82} C_VEL
LIN {X 0,Y 394.586,Z 935.928,A -85,B 0,C 180,E1 15973.471,E2 15973.471} C_VEL
LIN {X 0,Y 387.727,Z 950.733,A -85,B 0,C 180,E1 15971.314,E2 15971.314} C_VEL
LIN {X 0,Y 379.625,Z 967.832,A -85,B 0,C 180,E1 15968.433,E2 15968.433} C_VEL
LIN {X 0,Y 372.038,Z 983.339,A -85,B 0,C 180,E1 15965.298,E2 15965.298} C_VEL
LIN {X 0,Y 366.017,Z 995.796,A -85,B 0,C 180,E1 15962.373,E2 15962.373} C_VEL
LIN {X 0,Y 359.53,Z 1009.535,A -85,B 0,C 180,E1 15958.577,E2 15958.577} C_VEL
LIN {X 0,Y 354.703,Z 1020.248,A -85,B 0,C 180,E1 15955.014,E2 15955.014} C_VEL
LIN {X 0,Y 351.057,Z 1029.09,A -85,B 0,C 180,E1 15951.556,E2 15951.556} C_VEL
LIN {X 0,Y 347.644,Z 1038.508,A -85,B 0,C 180,E1 15947.06,E2 15947.06} C_VEL
LIN {X 0,Y 345.828,Z 1044.652,A -85,B 0,C 180,E1 15943.374,E2 15943.374} C_VEL
LIN {X 0,Y 344.77,Z 1049.351,A -85,B 0,C 180,E1 15939.852,E2 15939.852} C_VEL
LIN {X 0,Y 344.128,Z 1053.538,A -85,B 0,C 180,E1 15935.669,E2 15935.669} C_VEL
LIN {X 0,Y 343.932,Z 1055.876,A -85,B 0,C 180,E1 15931.833,E2 15931.833} C_VEL
LIN {X 0,Y 343.908,Z 1056.884,A -85,B 0,C 180,E1 15928.667,E2 15928.667} C_VEL
LIN {X 0,Y 343.909,Z 1056.989,A -85,B 0,C 180,E1 15925.33,E2 15925.33} C_VEL
LIN {X 0,Y 343.938,Z 1056.187,A -85,B 0,C 180,E1 15922.147,E2 15922.147} C_VEL
LIN {X 0,Y 344.091,Z 1054.491,A -85,B 0,C 180,E1 15918.943,E2 15918.943} C_VEL
LIN {X 0,Y 344.495,Z 1051.727,A -85,B 0,C 180,E1 15915.545,E2 15915.545} C_VEL
LIN {X 0,Y 345.584,Z 1047.113,A -85,B 0,C 180,E1 15911.442,E2 15911.442} C_VEL
LIN {X 0,Y 347.592,Z 1040.489,A -85,B 0,C 180,E1 15907.149,E2 15907.149} C_VEL
LIN {X 0,Y 350.058,Z 1033.968,A -85,B 0,C 180,E1 15903.722,E2 15903.722} C_VEL
LIN {X 0,Y 353.75,Z 1025.456,A -85,B 0,C 180,E1 15899.98,E2 15899.98} C_VEL
LIN {X 0,Y 359.279,Z 1013.793,A -85,B 0,C 180,E1 15895.794,E2 15895.794} C_VEL
LIN {X 0,Y 364.46,Z 1003.474,A -85,B 0,C 180,E1 15892.677,E2 15892.677} C_VEL
LIN {X 0,Y 366.39,Z 999.87,A -85,B 0,C 180,E1 15891.671,E2 15891.671} C_VEL
LIN {X 0,Y 367.521,Z 996.276,A -85,B 0,C 180,E1 15890.611,E2 15890.611} C_VEL
LIN {X 0,Y 367.513,Z 986.634,A -85,B 0,C 180,E1 15887.658,E2 15887.658} C_VEL
LIN {X 0,Y 368.811,Z 983.139,A -85,B 0,C 180,E1 15886.799,E2 15886.799} C_VEL
LIN {X 0,Y 377.313,Z 967.632,A -85,B 0,C 180,E1 15883.66,E2 15883.66} C_VEL
LIN {X 0,Y 386.283,Z 950.549,A -85,B 0,C 180,E1 15880.788,E2 15880.788} C_VEL
LIN {X 0,Y 394.038,Z 935.37,A -85,B 0,C 180,E1 15878.596,E2 15878.596} C_VEL
LIN {X 0,Y 403.432,Z 916.17,A -85,B 0,C 180,E1 15876.222,E2 15876.222} C_VEL
LIN {X 0,Y 412.252,Z 896.59,A -85,B 0,C 180,E1 15874.201,E2 15874.201} C_VEL
LIN {X 0,Y 419.72,Z 878.899,A -85,B 0,C 180,E1 15872.634,E2 15872.634} C_VEL
LIN {X 0,Y 428.127,Z 857.385,A -85,B 0,C 180,E1 15871.005,E2 15871.005} C_VEL
LIN {X 0,Y 435.84,Z 834.902,A -85,B 0,C 180,E1 15869.601,E2 15869.601} C_VEL
LIN {X 0,Y 441.78,Z 815.592,A -85,B 0,C 180,E1 15868.578,E2 15868.578} C_VEL
LIN {X 0,Y 448.228,Z 791.951,A -85,B 0,C 180,E1 15867.536,E2 15867.536} C_VEL
LIN {X 0,Y 453.87,Z 766.557,A -85,B 0,C 180,E1 15866.653,E2 15866.653} C_VEL
LIN {X 0,Y 457.67,Z 745.909,A -85,B 0,C 180,E1 15866.088,E2 15866.088} C_VEL
LIN {X 0,Y 461.204,Z 721.278,A -85,B 0,C 180,E1 15865.553,E2 15865.553} C_VEL
LIN {X 0,Y 464.488,Z 682.354,A -85,B 0,C 180,E1 15864.909,E2 15864.909} C_VEL
LIN {X 0,Y 481.088,Z 462.903,A -85,B 0,C 180,E1 15861.47,E2 15861.47} C_VEL
LIN {X 0,Y 473.426,Z 450.646,A -85,B 0,C 180,E1 15858.661,E2 15858.661} C_VEL
LIN {X 0,Y 468.141,Z 442.671,A -85,B 0,C 180,E1 15856.44,E2 15856.44} C_VEL
LIN {X 0,Y 463.248,Z 435.231,A -85,B 0,C 180,E1 15854.053,E2 15854.053} C_VEL
LIN {X 0,Y 459.386,Z 429.856,A -85,B 0,C 180,E1 15851.87,E2 15851.87} C_VEL
LIN {X 0,Y 456.217,Z 425.215,A -85,B 0,C 180,E1 15849.716,E2 15849.716} C_VEL
LIN {X 0,Y 453.204,Z 420.892,A -85,B 0,C 180,E1 15847.161,E2 15847.161} C_VEL
LIN {X 0,Y 452.395,Z 419.886,A -85,B 0,C 180,E1 15846.345,E2 15846.345} C_VEL
LIN {X 0,Y 449.82,Z 416.167,A -85,B 0,C 180,E1 15842.676,E2 15842.676} C_VEL
LIN {X 0,Y 449.37,Z 414.859,A -85,B 0,C 180,E1 15841.403,E2 15841.403} C_VEL
LIN {X 0,Y 449.039,Z 414.665,A -85,B 0,C 180,E1 15836.809,E2 15836.809} C_VEL
LIN {X 0,Y 449.569,Z 415.188,A -85,B 0,C 180,E1 15835.133,E2 15835.133} C_VEL
LIN {X 0,Y 451.823,Z 419.473,A -85,B 0,C 180,E1 15831.345,E2 15831.345} C_VEL
LIN {X 0,Y 453.181,Z 420.778,A -85,B 0,C 180,E1 15829.962,E2 15829.962} C_VEL
LIN {X 0,Y 456.446,Z 425.431,A -85,B 0,C 180,E1 15827.217,E2 15827.217} C_VEL
LIN {X 0,Y 460.893,Z 431.942,A -85,B 0,C 180,E1 15824.33,E2 15824.33} C_VEL
LIN {X 0,Y 464.476,Z 437.266,A -85,B 0,C 180,E1 15822.395,E2 15822.395} C_VEL
LIN {X 0,Y 469.665,Z 444.877,A -85,B 0,C 180,E1 15819.987,E2 15819.987} C_VEL
LIN {X 0,Y 475.495,Z 454.79,A -85,B 0,C 180,E1 15817.596,E2 15817.596} C_VEL
LIN {X 0,Y 481.031,Z 464.686,A -85,B 0,C 180,E1 15815.572,E2 15815.572} C_VEL
LIN {X 0,Y 463.835,Z 692.524,A -85,B 0,C 180,E1 15812.001,E2 15812.001} C_VEL
LIN {X 0,Y 460.718,Z 727.498,A -85,B 0,C 180,E1 15811.411,E2 15811.411} C_VEL
LIN {X 0,Y 457.326,Z 750.698,A -85,B 0,C 180,E1 15810.911,E2 15810.911} C_VEL
LIN {X 0,Y 453.163,Z 772.841,A -85,B 0,C 180,E1 15810.311,E2 15810.311} C_VEL
LIN {X 0,Y 446.88,Z 799.945,A -85,B 0,C 180,E1 15809.351,E2 15809.351} C_VEL
LIN {X 0,Y 441.106,Z 820.868,A -85,B 0,C 180,E1 15808.424,E2 15808.424} C_VEL
LIN {X 0,Y 435.03,Z 840.441,A -85,B 0,C 180,E1 15807.392,E2 15807.392} C_VEL
LIN {X 0,Y 426.801,Z 864.011,A -85,B 0,C 180,E1 15805.91,E2 15805.91} C_VEL
LIN {X 0,Y 418.844,Z 884.286,A -85,B 0,C 180,E1 15804.374,E2 15804.374} C_VEL
LIN {X 0,Y 411.222,Z 902.3,A -85,B 0,C 180,E1 15802.78,E2 15802.78} C_VEL
LIN {X 0,Y 401.774,Z 923.151,A -85,B 0,C 180,E1 15800.608,E2 15800.608} C_VEL
LIN {X 0,Y 393.102,Z 940.896,A -85,B 0,C 180,E1 15798.401,E2 15798.401} C_VEL
LIN {X 0,Y 385.269,Z 956.307,A -85,B 0,C 180,E1 15796.178,E2 15796.178} C_VEL
LIN {X 0,Y 376.275,Z 973.556,A -85,B 0,C 180,E1 15793.271,E2 15793.271} C_VEL
LIN {X 0,Y 368.202,Z 988.465,A -85,B 0,C 180,E1 15790.263,E2 15790.263} C_VEL
LIN {X 0,Y 361.407,Z 1001.097,A -85,B 0,C 180,E1 15787.293,E2 15787.293} C_VEL
LIN {X 0,Y 354.356,Z 1014.559,A -85,B 0,C 180,E1 15783.577,E2 15783.577} C_VEL
LIN {X 0,Y 348.531,Z 1025.967,A -85,B 0,C 180,E1 15779.756,E2 15779.756} C_VEL
LIN {X 0,Y 344.341,Z 1034.976,A -85,B 0,C 180,E1 15776.192,E2 15776.192} C_VEL
LIN {X 0,Y 340.481,Z 1044.297,A -85,B 0,C 180,E1 15771.717,E2 15771.717} C_VEL
LIN {X 0,Y 338.255,Z 1050.696,A -85,B 0,C 180,E1 15767.853,E2 15767.853} C_VEL
LIN {X 0,Y 336.967,Z 1055.484,A -85,B 0,C 180,E1 15764.258,E2 15764.258} C_VEL
LIN {X 0,Y 336.228,Z 1059.377,A -85,B 0,C 180,E1 15760.452,E2 15760.452} C_VEL
LIN {X 0,Y 335.945,Z 1062.256,A -85,B 0,C 180,E1 15756.224,E2 15756.224} C_VEL
LIN {X 0,Y 335.912,Z 1063.479,A -85,B 0,C 180,E1 15752.559,E2 15752.559} C_VEL
LIN {X 0,Y 335.913,Z 1063.613,A -85,B 0,C 180,E1 15749.147,E2 15749.147} C_VEL
LIN {X 0,Y 335.911,Z 1062.822,A -85,B 0,C 180,E1 15745.903,E2 15745.903} C_VEL
LIN {X 0,Y 336.004,Z 1061.008,A -85,B 0,C 180,E1 15742.476,E2 15742.476} C_VEL
LIN {X 0,Y 336.285,Z 1058.181,A -85,B 0,C 180,E1 15739.03,E2 15739.03} C_VEL
LIN {X 0,Y 337.188,Z 1053.482,A -85,B 0,C 180,E1 15734.874,E2 15734.874} C_VEL
LIN {X 0,Y 338.979,Z 1046.752,A -85,B 0,C 180,E1 15730.53,E2 15730.53} C_VEL
LIN {X 0,Y 341.228,Z 1040.149,A -85,B 0,C 180,E1 15727.063,E2 15727.063} C_VEL
LIN {X 0,Y 344.656,Z 1031.551,A -85,B 0,C 180,E1 15723.278,E2 15723.278} C_VEL
LIN {X 0,Y 349.877,Z 1019.742,A -85,B 0,C 180,E1 15719.021,E2 15719.021} C_VEL
LIN {X 0,Y 354.757,Z 1009.413,A -85,B 0,C 180,E1 15715.883,E2 15715.883} C_VEL
LIN {X 0,Y 360.878,Z 997.032,A -85,B 0,C 180,E1 15712.643,E2 15712.643} C_VEL
LIN {X 0,Y 368.775,Z 981.186,A -85,B 0,C 180,E1 15709.155,E2 15709.155} C_VEL
LIN {X 0,Y 375.919,Z 966.744,A -85,B 0,C 180,E1 15706.457,E2 15706.457} C_VEL
LIN {X 0,Y 384.125,Z 949.932,A -85,B 0,C 180,E1 15703.752,E2 15703.752} C_VEL
LIN {X 0,Y 393.069,Z 930.639,A -85,B 0,C 180,E1 15701.153,E2 15701.153} C_VEL
LIN {X 0,Y 400.598,Z 913.628,A -85,B 0,C 180,E1 15699.195,E2 15699.195} C_VEL
LIN {X 0,Y 409.132,Z 893.272,A -85,B 0,C 180,E1 15697.183,E2 15697.183} C_VEL
LIN {X 0,Y 417.205,Z 871.968,A -85,B 0,C 180,E1 15695.427,E2 15695.427} C_VEL
LIN {X 0,Y 423.833,Z 853.042,A -85,B 0,C 180,E1 15694.1,E2 15694.1} C_VEL
LIN {X 0,Y 430.684,Z 831.53,A -85,B 0,C 180,E1 15692.815,E2 15692.815} C_VEL
LIN {X 0,Y 437.399,Z 807.152,A -85,B 0,C 180,E1 15691.622,E2 15691.622} C_VEL
LIN {X 0,Y 442.115,Z 787.392,A -85,B 0,C 180,E1 15690.825,E2 15690.825} C_VEL
LIN {X 0,Y 446.596,Z 765.374,A -85,B 0,C 180,E1 15690.092,E2 15690.092} C_VEL
LIN {X 0,Y 451.142,Z 737.104,A -85,B 0,C 180,E1 15689.382,E2 15689.382} C_VEL
LIN {X 0,Y 453.64,Z 714.412,A -85,B 0,C 180,E1 15688.946,E2 15688.946} C_VEL
LIN {X 0,Y 469.82,Z 486.602,A -85,B 0,C 180,E1 15685.325,E2 15685.325} C_VEL
LIN {X 0,Y 471.773,Z 459.041,A -85,B 0,C 180,E1 15684.879,E2 15684.879} C_VEL
LIN {X 0,Y 465.293,Z 447.281,A -85,B 0,C 180,E1 15682.79,E2 15682.79} C_VEL
LIN {X 0,Y 459.668,Z 437.675,A -85,B 0,C 180,E1 15680.8,E2 15680.8} C_VEL
LIN {X 0,Y 452.869,Z 427.626,A -85,B 0,C 180,E1 15678.139,E2 15678.139} C_VEL
LIN {X 0,Y 447.329,Z 419.713,A -85,B 0,C 180,E1 15675.625,E2 15675.625} C_VEL
LIN {X 0,Y 444.078,Z 415.168,A -85,B 0,C 180,E1 15673.941,E2 15673.941} C_VEL
LIN {X 0,Y 440.759,Z 410.493,A -85,B 0,C 180,E1 15671.98,E2 15671.98} C_VEL
LIN {X 0,Y 437.21,Z 405.554,A -85,B 0,C 180,E1 15669.478,E2 15669.478} C_VEL
LIN {X 0,Y 434.042,Z 401.444,A -85,B 0,C 180,E1 15666.614,E2 15666.614} C_VEL
LIN {X 0,Y 433.392,Z 400.114,A -85,B 0,C 180,E1 15665.826,E2 15665.826} C_VEL
LIN {X 0,Y 430.256,Z 396.396,A -85,B 0,C 180,E1 15658.935,E2 15658.935} C_VEL
LIN {X 0,Y 430.458,Z 397.03,A -85,B 0,C 180,E1 15656.271,E2 15656.271} C_VEL
LIN {X 0,Y 433.631,Z 400.466,A -85,B 0,C 180,E1 15650.711,E2 15650.711} C_VEL
LIN {X 0,Y 436.09,Z 404.464,A -85,B 0,C 180,E1 15648.225,E2 15648.225} C_VEL
LIN {X 0,Y 437.743,Z 406.292,A -85,B 0,C 180,E1 15646.93,E2 15646.93} C_VEL
LIN {X 0,Y 441.125,Z 410.837,A -85,B 0,C 180,E1 15644.621,E2 15644.621} C_VEL
LIN {X 0,Y 445.789,Z 417.556,A -85,B 0,C 180,E1 15641.969,E2 15641.969} C_VEL
LIN {X 0,Y 449.897,Z 423.305,A -85,B 0,C 180,E1 15639.985,E2 15639.985} C_VEL
LIN {X 0,Y 454.893,Z 430.46,A -85,B 0,C 180,E1 15637.854,E2 15637.854} C_VEL
LIN {X 0,Y 463.306,Z 443.182,A -85,B 0,C 180,E1 15634.737,E2 15634.737} C_VEL
LIN {X 0,Y 471.608,Z 456.718,A -85,B 0,C 180,E1 15632.059,E2 15632.059} C_VEL
LIN {X 0,Y 471.841,Z 457.513,A -85,B 0,C 180,E1 15631.975,E2 15631.975} C_VEL
LIN {X 0,Y 456.005,Z 680.967,A -85,B 0,C 180,E1 15628.437,E2 15628.437} C_VEL
LIN {X 0,Y 452.854,Z 720.882,A -85,B 0,C 180,E1 15627.771,E2 15627.771} C_VEL
LIN {X 0,Y 449.435,Z 745.896,A -85,B 0,C 180,E1 15627.212,E2 15627.212} C_VEL
LIN {X 0,Y 445.853,Z 766.33,A -85,B 0,C 180,E1 15626.633,E2 15626.633} C_VEL
LIN {X 0,Y 440.64,Z 791.096,A -85,B 0,C 180,E1 15625.753,E2 15625.753} C_VEL
LIN {X 0,Y 434.454,Z 814.994,A -85,B 0,C 180,E1 15624.674,E2 15624.674} C_VEL
LIN {X 0,Y 428.62,Z 834.945,A -85,B 0,C 180,E1 15623.592,E2 15623.592} C_VEL
LIN {X 0,Y 421.04,Z 858.11,A -85,B 0,C 180,E1 15622.102,E2 15622.102} C_VEL
LIN {X 0,Y 413.108,Z 879.504,A -85,B 0,C 180,E1 15620.434,E2 15620.434} C_VEL
LIN {X 0,Y 405.953,Z 897.421,A -85,B 0,C 180,E1 15618.804,E2 15618.804} C_VEL
LIN {X 0,Y 397.323,Z 917.63,A -85,B 0,C 180,E1 15616.659,E2 15616.659} C_VEL
LIN {X 0,Y 388.722,Z 936.253,A -85,B 0,C 180,E1 15614.296,E2 15614.296} C_VEL
LIN {X 0,Y 381.2,Z 951.952,A -85,B 0,C 180,E1 15611.979,E2 15611.979} C_VEL
